LIN {X 0,Y 481.676,Z 380.486,A -85,B 0,C 180,E1 -6886.848,E2 -6886.848} C_VEL
LIN {X 0,Y 481.68,Z 380.488,A -85,B 0,C 180,E1 -6890.064,E2 -6890.064} C_VEL
LIN {X 0,Y 481.619,Z 380.495,A -85,B 0,C 180,E1 -6893.256,E2 -6893.256} C_VEL
LIN {X 0,Y 481.719,Z 380.64,A -85,B 0,C 180,E1 -6895.758,E2 -6895.758} C_VEL
LIN {X 0,Y 483.205,Z 388.494,A -85,B 0,C 180,E1 -6898.429,E2 -6898.429} C_VEL
LIN {X 0,Y 483.717,Z 393.145,A -85,B 0,C 180,E1 -6899.92,E2 -6899.92} C_VEL
LIN {X 0,Y 483.106,Z 403.096,A -85,B 0,C 180,E1 -6902.865,E2 -6902.865} C_VEL
LIN {X 0,Y 482.561,Z 413.944,A -85,B 0,C 180,E1 -6905.937,E2 -6905.937} C_VEL
LIN {X 0,Y 482.061,Z 425.792,A -85,B 0,C 180,E1 -6909.208,E2 -6909.208} C_VEL
LIN {X 0,Y 481.663,Z 438.463,A -85,B 0,C 180,E1 -6912.598,E2 -6912.598} C_VEL
LIN {X 0,Y 481.415,Z 448.444,A -85,B 0,C 180,E1 -6915.2,E2 -6915.2} C_VEL
LIN {X 0,Y 483.253,Z 462.341,A -85,B 0,C 180,E1 -6915.581,E2 -6915.581} C_VEL
LIN {X 0,Y 483.6,Z 467.954,A -85,B 0,C 180,E1 -6915.779,E2 -6915.779} C_VEL
LIN {X 0,Y 483.17,Z 480.671,A -85,B 0,C 180,E1 -6916.33,E2 -6916.33} C_VEL
LIN {X 0,Y 482.784,Z 492.217,A -85,B 0,C 180,E1 -6917.005,E2 -6917.005} C_VEL
LIN {X 0,Y 482.404,Z 503.568,A -85,B 0,C 180,E1 -6917.852,E2 -6917.852} C_VEL
LIN {X 0,Y 482.056,Z 513.298,A -85,B 0,C 180,E1 -6918.758,E2 -6918.758} C_VEL
LIN {X 0,Y 481.599,Z 523.341,A -85,B 0,C 180,E1 -6919.917,E2 -6919.917} C_VEL
LIN {X 0,Y 481.317,Z 532.179,A -85,B 0,C 180,E1 -6921.183,E2 -6921.183} C_VEL
LIN {X 0,Y 481.104,Z 539.214,A -85,B 0,C 180,E1 -6922.447,E2 -6922.447} C_VEL
LIN {X 0,Y 480.936,Z 545.233,A -85,B 0,C 180,E1 -6923.812,E2 -6923.812} C_VEL
LIN {X 0,Y 480.904,Z 549.252,A -85,B 0,C 180,E1 -6924.972,E2 -6924.972} C_VEL
LIN {X 0,Y 480.851,Z 551.584,A -85,B 0,C 180,E1 -6925.811,E2 -6925.811} C_VEL
LIN {X 0,Y 480.893,Z 553.484,A -85,B 0,C 180,E1 -6926.651,E2 -6926.651} C_VEL
LIN {X 0,Y 480.869,Z 554.904,A -85,B 0,C 180,E1 -6927.489,E2 -6927.489} C_VEL
LIN {X 0,Y 480.824,Z 555.914,A -85,B 0,C 180,E1 -6928.327,E2 -6928.327} C_VEL
LIN {X 0,Y 480.743,Z 556.751,A -85,B 0,C 180,E1 -6930.002,E2 -6930.002} C_VEL
LIN {X 0,Y 480.825,Z 555.927,A -85,B 0,C 180,E1 -6931.677,E2 -6931.677} C_VEL
LIN {X 0,Y 480.87,Z 554.926,A -85,B 0,C 180,E1 -6932.515,E2 -6932.515} C_VEL
LIN {X 0,Y 480.894,Z 553.512,A -85,B 0,C 180,E1 -6933.353,E2 -6933.353} C_VEL
LIN {X 0,Y 480.847,Z 550.542,A -85,B 0,C 180,E1 -6934.613,E2 -6934.613} C_VEL
LIN {X 0,Y 480.952,Z 546.523,A -85,B 0,C 180,E1 -6935.873,E2 -6935.873} C_VEL
LIN {X 0,Y 481.11,Z 540.312,A -85,B 0,C 180,E1 -6937.345,E2 -6937.345} C_VEL
LIN {X 0,Y 481.308,Z 533.534,A -85,B 0,C 180,E1 -6938.609,E2 -6938.609} C_VEL
LIN {X 0,Y 481.557,Z 525.1,A -85,B 0,C 180,E1 -6939.876,E2 -6939.876} C_VEL
LIN {X 0,Y 481.935,Z 516.392,A -85,B 0,C 180,E1 -6940.93,E2 -6940.93} C_VEL
LIN {X 0,Y 482.315,Z 505.902,A -85,B 0,C 180,E1 -6941.963,E2 -6941.963} C_VEL
LIN {X 0,Y 482.683,Z 495.234,A -85,B 0,C 180,E1 -6942.809,E2 -6942.809} C_VEL
LIN {X 0,Y 483.131,Z 482.915,A -85,B 0,C 180,E1 -6943.568,E2 -6943.568} C_VEL
LIN {X 0,Y 483.542,Z 470.344,A -85,B 0,C 180,E1 -6944.146,E2 -6944.146} C_VEL
LIN {X 0,Y 483.49,Z 464.03,A -85,B 0,C 180,E1 -6944.375,E2 -6944.375} C_VEL
LIN {X 0,Y 481.762,Z 451.22,A -85,B 0,C 180,E1 -6944.751,E2 -6944.751} C_VEL
LIN {X 0,Y 481.415,Z 448.546,A -85,B 0,C 180,E1 -6944.83,E2 -6944.83} C_VEL
LIN {X 0,Y 481.748,Z 435.725,A -85,B 0,C 180,E1 -6948.186,E2 -6948.186} C_VEL
LIN {X 0,Y 482.152,Z 423.863,A -85,B 0,C 180,E1 -6951.373,E2 -6951.373} C_VEL
LIN {X 0,Y 482.662,Z 412.396,A -85,B 0,C 180,E1 -6954.52,E2 -6954.52} C_VEL
LIN {X 0,Y 483.215,Z 401.049,A -85,B 0,C 180,E1 -6957.738,E2 -6957.738} C_VEL
LIN {X 0,Y 483.662,Z 393.005,A -85,B 0,C 180,E1 -6960.088,E2 -6960.088} C_VEL
LIN {X 0,Y 483.172,Z 388.19,A -85,B 0,C 180,E1 -6961.578,E2 -6961.578} C_VEL
LIN {X 0,Y 481.724,Z 380.48,A -85,B 0,C 180,E1 -6964.174,E2 -6964.174} C_VEL
LIN {X 0,Y 481.63,Z 380.493,A -85,B 0,C 180,E1 -6967.798,E2 -6967.798} C_VEL
LIN {X 0,Y 481.643,Z 380.488,A -85,B 0,C 180,E1 -6970.644,E2 -6970.644} C_VEL
LIN {X 0,Y 481.619,Z 380.494,A -85,B 0,C 180,E1 -6973.303,E2 -6973.303} C_VEL
LIN {X 0,Y 481.658,Z 380.486,A -85,B 0,C 180,E1 -6975.642,E2 -6975.642} C_VEL
LIN {X 0,Y 481.632,Z 380.49,A -85,B 0,C 180,E1 -6978.955,E2 -6978.955} C_VEL
LIN {X 0,Y 481.659,Z 380.484,A -85,B 0,C 180,E1 -6981.993,E2 -6981.993} C_VEL
LIN {X 0,Y 481.689,Z 380.481,A -85,B 0,C 180,E1 -6985.318,E2 -6985.318} C_VEL
LIN {X 0,Y 481.647,Z 380.488,A -85,B 0,C 180,E1 -6988.311,E2 -6988.311} C_VEL
LIN {X 0,Y 481.663,Z 380.488,A -85,B 0,C 180,E1 -6991.216,E2 -6991.216} C_VEL
LIN {X 0,Y 481.621,Z 380.49,A -85,B 0,C 180,E1 -6994.038,E2 -6994.038} C_VEL
LIN {X 0,Y 481.658,Z 380.491,A -85,B 0,C 180,E1 -6996.818,E2 -6996.818} C_VEL
LIN {X 0,Y 481.7,Z 380.481,A -85,B 0,C 180,E1 -6999.503,E2 -6999.503} C_VEL
LIN {X 0,Y 481.709,Z 380.485,A -85,B 0,C 180,E1 -7002.158,E2 -7002.158} C_VEL
LIN {X 0,Y 481.747,Z 380.476,A -85,B 0,C 180,E1 -7004.776,E2 -7004.776} C_VEL
LIN {X 0,Y 481.754,Z 380.476,A -85,B 0,C 180,E1 -7008.215,E2 -7008.215} C_VEL
LIN {X 0,Y 481.719,Z 380.481,A -85,B 0,C 180,E1 -7011.611,E2 -7011.611} C_VEL
LIN {X 0,Y 481.781,Z 380.473,A -85,B 0,C 180,E1 -7014.139,E2 -7014.139} C_VEL
LIN {X 0,Y 481.503,Z 380.649,A -85,B 0,C 180,E1 -7016.967,E2 -7016.967} C_VEL
LIN {X 0,Y 481.645,Z 387.989,A -85,B 0,C 180,E1 -7020,E2 -7020} C_VEL
LIN {X 0,Y 481.317,Z 393.994,A -85,B 0,C 180,E1 -7022.51,E2 -7022.51} C_VEL
LIN {X 0,Y 481.398,Z 399.763,A -85,B 0,C 180,E1 -7025.025,E2 -7025.025} C_VEL
LIN {X 0,Y 481.34,Z 405.639,A -85,B 0,C 180,E1 -7027.551,E2 -7027.551} C_VEL
LIN {X 0,Y 481.25,Z 413.309,A -85,B 0,C 180,E1 -7030.944,E2 -7030.944} C_VEL
LIN {X 0,Y 481.1,Z 420.994,A -85,B 0,C 180,E1 -7034.379,E2 -7034.379} C_VEL
LIN {X 0,Y 481.05,Z 424.92,A -85,B 0,C 180,E1 -7036.143,E2 -7036.143} C_VEL
LIN {X 0,Y 483.616,Z 438.35,A -85,B 0,C 180,E1 -7036.597,E2 -7036.597} C_VEL
LIN {X 0,Y 483.92,Z 441.544,A -85,B 0,C 180,E1 -7036.722,E2 -7036.722} C_VEL
LIN {X 0,Y 483.588,Z 454.148,A -85,B 0,C 180,E1 -7037.278,E2 -7037.278} C_VEL
LIN {X 0,Y 483.157,Z 464.801,A -85,B 0,C 180,E1 -7037.895,E2 -7037.895} C_VEL
LIN {X 0,Y 482.794,Z 475.459,A -85,B 0,C 180,E1 -7038.678,E2 -7038.678} C_VEL
LIN {X 0,Y 482.35,Z 486.451,A -85,B 0,C 180,E1 -7039.69,E2 -7039.69} C_VEL
LIN {X 0,Y 481.93,Z 495.839,A -85,B 0,C 180,E1 -7040.757,E2 -7040.757} C_VEL
LIN {X 0,Y 481.61,Z 503.654,A -85,B 0,C 180,E1 -7041.846,E2 -7041.846} C_VEL
LIN {X 0,Y 481.338,Z 511.583,A -85,B 0,C 180,E1 -7043.217,E2 -7043.217} C_VEL
LIN {X 0,Y 481.031,Z 517.926,A -85,B 0,C 180,E1 -7044.602,E2 -7044.602} C_VEL
LIN {X 0,Y 480.953,Z 522.785,A -85,B 0,C 180,E1 -7046,E2 -7046} C_VEL
LIN {X 0,Y 480.834,Z 526.37,A -85,B 0,C 180,E1 -7047.413,E2 -7047.413} C_VEL
LIN {X 0,Y 480.752,Z 528.76,A -85,B 0,C 180,E1 -7048.843,E2 -7048.843} C_VEL
LIN {X 0,Y 480.729,Z 530.029,A -85,B 0,C 180,E1 -7050.395,E2 -7050.395} C_VEL
LIN {X 0,Y 480.712,Z 529.851,A -85,B 0,C 180,E1 -7052.008,E2 -7052.008} C_VEL
LIN {X 0,Y 480.744,Z 528.314,A -85,B 0,C 180,E1 -7053.561,E2 -7053.561} C_VEL
LIN {X 0,Y 480.831,Z 525.481,A -85,B 0,C 180,E1 -7055.062,E2 -7055.062} C_VEL
LIN {X 0,Y 480.977,Z 521.357,A -85,B 0,C 180,E1 -7056.518,E2 -7056.518} C_VEL
LIN {X 0,Y 481.115,Z 516.002,A -85,B 0,C 180,E1 -7057.924,E2 -7057.924} C_VEL
LIN {X 0,Y 481.368,Z 509.214,A -85,B 0,C 180,E1 -7059.302,E2 -7059.302} C_VEL
LIN {X 0,Y 481.699,Z 500.773,A -85,B 0,C 180,E1 -7060.651,E2 -7060.651} C_VEL
LIN {X 0,Y 482.022,Z 492.106,A -85,B 0,C 180,E1 -7061.771,E2 -7061.771} C_VEL
LIN {X 0,Y 482.459,Z 482.471,A -85,B 0,C 180,E1 -7062.78,E2 -7062.78} C_VEL
LIN {X 0,Y 482.875,Z 471.084,A -85,B 0,C 180,E1 -7063.744,E2 -7063.744} C_VEL
LIN {X 0,Y 483.301,Z 460.089,A -85,B 0,C 180,E1 -7064.479,E2 -7064.479} C_VEL
LIN {X 0,Y 483.712,Z 448.856,A -85,B 0,C 180,E1 -7065.06,E2 -7065.06} C_VEL
LIN {X 0,Y 483.741,Z 439.076,A -85,B 0,C 180,E1 -7065.458,E2 -7065.458} C_VEL
LIN {X 0,Y 481.378,Z 426.409,A -85,B 0,C 180,E1 -7065.891,E2 -7065.891} C_VEL
LIN {X 0,Y 481.036,Z 424.605,A -85,B 0,C 180,E1 -7065.96,E2 -7065.96} C_VEL
LIN {X 0,Y 481.132,Z 418.161,A -85,B 0,C 180,E1 -7068.903,E2 -7068.903} C_VEL
LIN {X 0,Y 481.192,Z 411.015,A -85,B 0,C 180,E1 -7072.161,E2 -7072.161} C_VEL
LIN {X 0,Y 481.33,Z 404.161,A -85,B 0,C 180,E1 -7075.287,E2 -7075.287} C_VEL
LIN {X 0,Y 481.362,Z 403.419,A -85,B 0,C 180,E1 -7075.624,E2 -7075.624} C_VEL
LIN {X 0,Y 480.754,Z 402.002,A -85,B 0,C 180,E1 -7076.302,E2 -7076.302} C_VEL
LIN {X 0,Y 477.91,Z 399.902,A -85,B 0,C 180,E1 -7077.409,E2 -7077.409} C_VEL
LIN {X 0,Y 475.496,Z 398.224,A -85,B 0,C 180,E1 -7078.302,E2 -7078.302} C_VEL
LIN {X 0,Y 474.494,Z 396.844,A -85,B 0,C 180,E1 -7078.99,E2 -7078.99} C_VEL
LIN {X 0,Y 474.432,Z 396.349,A -85,B 0,C 180,E1 -7079.221,E2 -7079.221} C_VEL
LIN {X 0,Y 474.464,Z 389.854,A -85,B 0,C 180,E1 -7082.185,E2 -7082.185} C_VEL
LIN {X 0,Y 474.646,Z 382.584,A -85,B 0,C 180,E1 -7085.505,E2 -7085.505} C_VEL
LIN {X 0,Y 474.683,Z 381.36,A -85,B 0,C 180,E1 -7086.088,E2 -7086.088} C_VEL
LIN {X 0,Y 474.673,Z 381.359,A -85,B 0,C 180,E1 -7089.184,E2 -7089.184} C_VEL
LIN {X 0,Y 474.646,Z 381.364,A -85,B 0,C 180,E1 -7091.882,E2 -7091.882} C_VEL
LIN {X 0,Y 474.702,Z 381.353,A -85,B 0,C 180,E1 -7094.543,E2 -7094.543} C_VEL
LIN {X 0,Y 474.705,Z 381.355,A -85,B 0,C 180,E1 -7098.036,E2 -7098.036} C_VEL
LIN {X 0,Y 474.727,Z 381.355,A -85,B 0,C 180,E1 -7101.485,E2 -7101.485} C_VEL
LIN {X 0,Y 474.743,Z 381.352,A -85,B 0,C 180,E1 -7104.902,E2 -7104.902} C_VEL
LIN {X 0,Y 474.874,Z 381.335,A -85,B 0,C 180,E1 -7107.453,E2 -7107.453} C_VEL
LIN {X 0,Y 474.91,Z 381.45,A -85,B 0,C 180,E1 -7109.892,E2 -7109.892} C_VEL
LIN {X 0,Y 474.733,Z 386.231,A -85,B 0,C 180,E1 -7112.544,E2 -7112.544} C_VEL
LIN {X 0,Y 474.574,Z 392.513,A -85,B 0,C 180,E1 -7115.948,E2 -7115.948} C_VEL
LIN {X 0,Y 474.425,Z 397.306,A -85,B 0,C 180,E1 -7118.517,E2 -7118.517} C_VEL
LIN {X 0,Y 474.306,Z 403.992,A -85,B 0,C 180,E1 -7122.056,E2 -7122.056} C_VEL
LIN {X 0,Y 474.1,Z 410.649,A -85,B 0,C 180,E1 -7125.518,E2 -7125.518} C_VEL
LIN {X 0,Y 473.939,Z 417.514,A -85,B 0,C 180,E1 -7129.038,E2 -7129.038} C_VEL
LIN {X 0,Y 473.922,Z 421.247,A -85,B 0,C 180,E1 -7130.937,E2 -7130.937} C_VEL
LIN {X 0,Y 475.816,Z 432.165,A -85,B 0,C 180,E1 -7131.36,E2 -7131.36} C_VEL
LIN {X 0,Y 476.036,Z 438.597,A -85,B 0,C 180,E1 -7131.657,E2 -7131.657} C_VEL
LIN {X 0,Y 475.665,Z 448.951,A -85,B 0,C 180,E1 -7132.245,E2 -7132.245} C_VEL
LIN {X 0,Y 475.314,Z 458.419,A -85,B 0,C 180,E1 -7132.951,E2 -7132.951} C_VEL
LIN {X 0,Y 474.982,Z 468.268,A -85,B 0,C 180,E1 -7133.892,E2 -7133.892} C_VEL
LIN {X 0,Y 474.64,Z 477.014,A -85,B 0,C 180,E1 -7134.958,E2 -7134.958} C_VEL
LIN {X 0,Y 474.346,Z 484.62,A -85,B 0,C 180,E1 -7136.151,E2 -7136.151} C_VEL
LIN {X 0,Y 474.047,Z 490.599,A -85,B 0,C 180,E1 -7137.358,E2 -7137.358} C_VEL
LIN {X 0,Y 473.984,Z 495.44,A -85,B 0,C 180,E1 -7138.65,E2 -7138.65} C_VEL
LIN {X 0,Y 473.866,Z 498.551,A -85,B 0,C 180,E1 -7139.788,E2 -7139.788} C_VEL
LIN {X 0,Y 473.714,Z 501.15,A -85,B 0,C 180,E1 -7141.279,E2 -7141.279} C_VEL
LIN {X 0,Y 473.679,Z 502.019,A -85,B 0,C 180,E1 -7142.282,E2 -7142.282} C_VEL
LIN {X 0,Y 473.693,Z 502.038,A -85,B 0,C 180,E1 -7143.814,E2 -7143.814} C_VEL
LIN {X 0,Y 473.799,Z 500.472,A -85,B 0,C 180,E1 -7145.342,E2 -7145.342} C_VEL
LIN {X 0,Y 473.948,Z 497.426,A -85,B 0,C 180,E1 -7146.799,E2 -7146.799} C_VEL
LIN {X 0,Y 474.043,Z 494.299,A -85,B 0,C 180,E1 -7147.824,E2 -7147.824} C_VEL
LIN {X 0,Y 474.216,Z 489.417,A -85,B 0,C 180,E1 -7149.036,E2 -7149.036} C_VEL
LIN {X 0,Y 474.438,Z 483.837,A -85,B 0,C 180,E1 -7150.115,E2 -7150.115} C_VEL
LIN {X 0,Y 474.683,Z 477.63,A -85,B 0,C 180,E1 -7151.084,E2 -7151.084} C_VEL
LIN {X 0,Y 474.927,Z 470.21,A -85,B 0,C 180,E1 -7152.025,E2 -7152.025} C_VEL
LIN {X 0,Y 475.324,Z 460.576,A -85,B 0,C 180,E1 -7152.993,E2 -7152.993} C_VEL
LIN {X 0,Y 475.726,Z 451.213,A -85,B 0,C 180,E1 -7153.726,E2 -7153.726} C_VEL
LIN {X 0,Y 476.046,Z 440.21,A -85,B 0,C 180,E1 -7154.39,E2 -7154.39} C_VEL
LIN {X 0,Y 475.974,Z 432.535,A -85,B 0,C 180,E1 -7154.746,E2 -7154.746} C_VEL
LIN {X 0,Y 473.94,Z 421.51,A -85,B 0,C 180,E1 -7155.188,E2 -7155.188} C_VEL
LIN {X 0,Y 474.031,Z 415.761,A -85,B 0,C 180,E1 -7158.151,E2 -7158.151} C_VEL
LIN {X 0,Y 474.098,Z 409.341,A -85,B 0,C 180,E1 -7161.494,E2 -7161.494} C_VEL
LIN {X 0,Y 474.207,Z 405.279,A -85,B 0,C 180,E1 -7163.643,E2 -7163.643} C_VEL
LIN {X 0,Y 474.346,Z 399.44,A -85,B 0,C 180,E1 -7166.757,E2 -7166.757} C_VEL
LIN {X 0,Y 474.483,Z 393.793,A -85,B 0,C 180,E1 -7169.762,E2 -7169.762} C_VEL
LIN {X 0,Y 474.692,Z 388.447,A -85,B 0,C 180,E1 -7172.68,E2 -7172.68} C_VEL
LIN {X 0,Y 474.819,Z 383.281,A -85,B 0,C 180,E1 -7175.516,E2 -7175.516} C_VEL
LIN {X 0,Y 474.697,Z 381.36,A -85,B 0,C 180,E1 -7176.617,E2 -7176.617} C_VEL
LIN {X 0,Y 474.633,Z 381.365,A -85,B 0,C 180,E1 -7180.089,E2 -7180.089} C_VEL
LIN {X 0,Y 474.627,Z 381.367,A -85,B 0,C 180,E1 -7182.774,E2 -7182.774} C_VEL
LIN {X 0,Y 474.63,Z 381.365,A -85,B 0,C 180,E1 -7185.421,E2 -7185.421} C_VEL
LIN {X 0,Y 474.719,Z 381.353,A -85,B 0,C 180,E1 -7188.038,E2 -7188.038} C_VEL
LIN {X 0,Y 474.711,Z 381.355,A -85,B 0,C 180,E1 -7191.486,E2 -7191.486} C_VEL
LIN {X 0,Y 474.769,Z 381.348,A -85,B 0,C 180,E1 -7194.053,E2 -7194.053} C_VEL
LIN {X 0,Y 474.88,Z 381.333,A -85,B 0,C 180,E1 -7197.456,E2 -7197.456} C_VEL
LIN {X 0,Y 474.886,Z 381.332,A -85,B 0,C 180,E1 -7200,E2 -7200} C_VEL
LIN {X 0,Y 474.88,Z 381.332,A -85,B 0,C 180,E1 -7202.545,E2 -7202.545} C_VEL
LIN {X 0,Y 474.77,Z 381.347,A -85,B 0,C 180,E1 -7205.948,E2 -7205.948} C_VEL
LIN {X 0,Y 474.707,Z 381.357,A -85,B 0,C 180,E1 -7208.514,E2 -7208.514} C_VEL
LIN {X 0,Y 474.72,Z 381.351,A -85,B 0,C 180,E1 -7211.962,E2 -7211.962} C_VEL
LIN {X 0,Y 474.68,Z 381.356,A -85,B 0,C 180,E1 -7215.779,E2 -7215.779} C_VEL
LIN {X 0,Y 474.646,Z 381.36,A -85,B 0,C 180,E1 -7219.011,E2 -7219.011} C_VEL
LIN {X 0,Y 474.623,Z 381.363,A -85,B 0,C 180,E1 -7221.728,E2 -7221.728} C_VEL
LIN {X 0,Y 474.641,Z 381.361,A -85,B 0,C 180,E1 -7224.494,E2 -7224.494} C_VEL
LIN {X 0,Y 474.678,Z 381.357,A -85,B 0,C 180,E1 -7227.34,E2 -7227.34} C_VEL
LIN {X 0,Y 474.59,Z 381.368,A -85,B 0,C 180,E1 -7230.813,E2 -7230.813} C_VEL
LIN {X 0,Y 474.62,Z 381.367,A -85,B 0,C 180,E1 -7233.986,E2 -7233.986} C_VEL
LIN {X 0,Y 474.559,Z 381.375,A -85,B 0,C 180,E1 -7236.902,E2 -7236.902} C_VEL
LIN {X 0,Y 474.638,Z 381.364,A -85,B 0,C 180,E1 -7239.654,E2 -7239.654} C_VEL
LIN {X 0,Y 474.637,Z 381.364,A -85,B 0,C 180,E1 -7242.932,E2 -7242.932} C_VEL
LIN {X 0,Y 474.604,Z 381.368,A -85,B 0,C 180,E1 -7245.898,E2 -7245.898} C_VEL
LIN {X 0,Y 474.633,Z 381.365,A -85,B 0,C 180,E1 -7249.041,E2 -7249.041} C_VEL
LIN {X 0,Y 474.608,Z 381.368,A -85,B 0,C 180,E1 -7251.705,E2 -7251.705} C_VEL
LIN {X 0,Y 474.653,Z 381.381,A -85,B 0,C 180,E1 -7255.394,E2 -7255.394} C_VEL
LIN {X 0,Y 476.288,Z 390.069,A -85,B 0,C 180,E1 -7258.409,E2 -7258.409} C_VEL
LIN {X 0,Y 476.747,Z 394.694,A -85,B 0,C 180,E1 -7259.923,E2 -7259.923} C_VEL
LIN {X 0,Y 476.124,Z 404.14,A -85,B 0,C 180,E1 -7262.771,E2 -7262.771} C_VEL
LIN {X 0,Y 475.535,Z 415.372,A -85,B 0,C 180,E1 -7266.023,E2 -7266.023} C_VEL
LIN {X 0,Y 475.017,Z 426.749,A -85,B 0,C 180,E1 -7269.204,E2 -7269.204} C_VEL
LIN {X 0,Y 474.614,Z 438.219,A -85,B 0,C 180,E1 -7272.331,E2 -7272.331} C_VEL
LIN {X 0,Y 474.366,Z 448.416,A -85,B 0,C 180,E1 -7275.003,E2 -7275.003} C_VEL
LIN {X 0,Y 476.165,Z 462.258,A -85,B 0,C 180,E1 -7275.389,E2 -7275.389} C_VEL
LIN {X 0,Y 476.669,Z 467.857,A -85,B 0,C 180,E1 -7275.596,E2 -7275.596} C_VEL
LIN {X 0,Y 476.268,Z 480.007,A -85,B 0,C 180,E1 -7276.128,E2 -7276.128} C_VEL
LIN {X 0,Y 475.802,Z 492.581,A -85,B 0,C 180,E1 -7276.876,E2 -7276.876} C_VEL
LIN {X 0,Y 475.375,Z 503.595,A -85,B 0,C 180,E1 -7277.718,E2 -7277.718} C_VEL
LIN {X 0,Y 475.005,Z 513.788,A -85,B 0,C 180,E1 -7278.697,E2 -7278.697} C_VEL
LIN {X 0,Y 474.562,Z 522.866,A -85,B 0,C 180,E1 -7279.766,E2 -7279.766} C_VEL
LIN {X 0,Y 474.258,Z 531.723,A -85,B 0,C 180,E1 -7281.051,E2 -7281.051} C_VEL
LIN {X 0,Y 474.034,Z 538.776,A -85,B 0,C 180,E1 -7282.334,E2 -7282.334} C_VEL
LIN {X 0,Y 473.848,Z 544.281,A -85,B 0,C 180,E1 -7283.582,E2 -7283.582} C_VEL
LIN {X 0,Y 473.838,Z 548.833,A -85,B 0,C 180,E1 -7284.896,E2 -7284.896} C_VEL
LIN {X 0,Y 473.754,Z 551.167,A -85,B 0,C 180,E1 -7285.748,E2 -7285.748} C_VEL
LIN {X 0,Y 473.819,Z 553.072,A -85,B 0,C 180,E1 -7286.601,E2 -7286.601} C_VEL
LIN {X 0,Y 473.783,Z 554.495,A -85,B 0,C 180,E1 -7287.451,E2 -7287.451} C_VEL
LIN {X 0,Y 473.758,Z 555.508,A -85,B 0,C 180,E1 -7288.302,E2 -7288.302} C_VEL
LIN {X 0,Y 473.67,Z 556.348,A -85,B 0,C 180,E1 -7290.002,E2 -7290.002} C_VEL
LIN {X 0,Y 473.758,Z 555.525,A -85,B 0,C 180,E1 -7291.702,E2 -7291.702} C_VEL
LIN {X 0,Y 473.784,Z 554.522,A -85,B 0,C 180,E1 -7292.552,E2 -7292.552} C_VEL
LIN {X 0,Y 473.82,Z 553.106,A -85,B 0,C 180,E1 -7293.403,E2 -7293.403} C_VEL
LIN {X 0,Y 473.77,Z 550.134,A -85,B 0,C 180,E1 -7294.682,E2 -7294.682} C_VEL
LIN {X 0,Y 473.856,Z 546.108,A -85,B 0,C 180,E1 -7295.961,E2 -7295.961} C_VEL
LIN {X 0,Y 474.019,Z 539.889,A -85,B 0,C 180,E1 -7297.456,E2 -7297.456} C_VEL
LIN {X 0,Y 474.235,Z 533.101,A -85,B 0,C 180,E1 -7298.739,E2 -7298.739} C_VEL
LIN {X 0,Y 474.497,Z 524.644,A -85,B 0,C 180,E1 -7300.024,E2 -7300.024} C_VEL
LIN {X 0,Y 474.892,Z 515.912,A -85,B 0,C 180,E1 -7301.094,E2 -7301.094} C_VEL
LIN {X 0,Y 475.283,Z 505.622,A -85,B 0,C 180,E1 -7302.121,E2 -7302.121} C_VEL
LIN {X 0,Y 475.737,Z 494.376,A -85,B 0,C 180,E1 -7303.021,E2 -7303.021} C_VEL
LIN {X 0,Y 476.195,Z 482.263,A -85,B 0,C 180,E1 -7303.769,E2 -7303.769} C_VEL
LIN {X 0,Y 476.613,Z 469.574,A -85,B 0,C 180,E1 -7304.356,E2 -7304.356} C_VEL
LIN {X 0,Y 476.524,Z 464.706,A -85,B 0,C 180,E1 -7304.536,E2 -7304.536} C_VEL
LIN {X 0,Y 474.842,Z 451.844,A -85,B 0,C 180,E1 -7304.934,E2 -7304.934} C_VEL
LIN {X 0,Y 474.366,Z 448.348,A -85,B 0,C 180,E1 -7305.028,E2 -7305.028} C_VEL
LIN {X 0,Y 474.71,Z 435.803,A -85,B 0,C 180,E1 -7308.387,E2 -7308.387} C_VEL
LIN {X 0,Y 475.154,Z 423.664,A -85,B 0,C 180,E1 -7311.703,E2 -7311.703} C_VEL
LIN {X 0,Y 475.712,Z 412.251,A -85,B 0,C 180,E1 -7314.902,E2 -7314.902} C_VEL
LIN {X 0,Y 476.342,Z 400.942,A -85,B 0,C 180,E1 -7318.174,E2 -7318.174} C_VEL
LIN {X 0,Y 476.705,Z 394.535,A -85,B 0,C 180,E1 -7320.085,E2 -7320.085} C_VEL
LIN {X 0,Y 476.251,Z 389.742,A -85,B 0,C 180,E1 -7321.593,E2 -7321.593} C_VEL
LIN {X 0,Y 474.685,Z 381.356,A -85,B 0,C 180,E1 -7324.431,E2 -7324.431} C_VEL
LIN {X 0,Y 474.591,Z 381.368,A -85,B 0,C 180,E1 -7327.385,E2 -7327.385} C_VEL
LIN {X 0,Y 474.611,Z 381.368,A -85,B 0,C 180,E1 -7329.645,E2 -7329.645} C_VEL
LIN {X 0,Y 474.571,Z 381.37,A -85,B 0,C 180,E1 -7332.94,E2 -7332.94} C_VEL
LIN {X 0,Y 474.608,Z 381.361,A -85,B 0,C 180,E1 -7335.895,E2 -7335.895} C_VEL
LIN {X 0,Y 474.607,Z 381.365,A -85,B 0,C 180,E1 -7339.045,E2 -7339.045} C_VEL
LIN {X 0,Y 474.615,Z 381.36,A -85,B 0,C 180,E1 -7341.705,E2 -7341.705} C_VEL
LIN {X 0,Y 474.629,Z 381.363,A -85,B 0,C 180,E1 -7344.726,E2 -7344.726} C_VEL
LIN {X 0,Y 474.633,Z 381.365,A -85,B 0,C 180,E1 -7347.787,E2 -7347.787} C_VEL
LIN {X 0,Y 474.603,Z 381.365,A -85,B 0,C 180,E1 -7350.891,E2 -7350.891} C_VEL
LIN {X 0,Y 474.575,Z 381.371,A -85,B 0,C 180,E1 -7353.623,E2 -7353.623} C_VEL
LIN {X 0,Y 474.639,Z 381.363,A -85,B 0,C 180,E1 -7356.642,E2 -7356.642} C_VEL
LIN {X 0,Y 474.659,Z 381.36,A -85,B 0,C 180,E1 -7360.089,E2 -7360.089} C_VEL
LIN {X 0,Y 474.653,Z 381.361,A -85,B 0,C 180,E1 -7362.774,E2 -7362.774} C_VEL
LIN {X 0,Y 474.651,Z 381.362,A -85,B 0,C 180,E1 -7365.421,E2 -7365.421} C_VEL
LIN {X 0,Y 474.708,Z 381.355,A -85,B 0,C 180,E1 -7368.037,E2 -7368.037} C_VEL
LIN {X 0,Y 474.669,Z 381.361,A -85,B 0,C 180,E1 -7371.485,E2 -7371.485} C_VEL
LIN {X 0,Y 474.744,Z 381.349,A -85,B 0,C 180,E1 -7374.052,E2 -7374.052} C_VEL
LIN {X 0,Y 474.572,Z 381.371,A -85,B 0,C 180,E1 -7375.753,E2 -7375.753} C_VEL
LIN {X 0,Y 474.482,Z 381.56,A -85,B 0,C 180,E1 -7376.922,E2 -7376.922} C_VEL
LIN {X 0,Y 474.627,Z 387.942,A -85,B 0,C 180,E1 -7379.576,E2 -7379.576} C_VEL
LIN {X 0,Y 474.345,Z 393.996,A -85,B 0,C 180,E1 -7382.122,E2 -7382.122} C_VEL
LIN {X 0,Y 474.348,Z 400.847,A -85,B 0,C 180,E1 -7385.1,E2 -7385.1} C_VEL
LIN {X 0,Y 474.278,Z 406.608,A -85,B 0,C 180,E1 -7387.664,E2 -7387.664} C_VEL
LIN {X 0,Y 474.198,Z 414.433,A -85,B 0,C 180,E1 -7391.108,E2 -7391.108} C_VEL
LIN {X 0,Y 474.029,Z 422.187,A -85,B 0,C 180,E1 -7394.598,E2 -7394.598} C_VEL
LIN {X 0,Y 473.98,Z 425.118,A -85,B 0,C 180,E1 -7395.921,E2 -7395.921} C_VEL
LIN {X 0,Y 476.607,Z 438.496,A -85,B 0,C 180,E1 -7396.38,E2 -7396.38} C_VEL
LIN {X 0,Y 477.035,Z 442.309,A -85,B 0,C 180,E1 -7396.536,E2 -7396.536} C_VEL
LIN {X 0,Y 476.662,Z 454.69,A -85,B 0,C 180,E1 -7397.095,E2 -7397.095} C_VEL
LIN {X 0,Y 476.176,Z 466.887,A -85,B 0,C 180,E1 -7397.833,E2 -7397.833} C_VEL
LIN {X 0,Y 475.702,Z 478.517,A -85,B 0,C 180,E1 -7398.743,E2 -7398.743} C_VEL
LIN {X 0,Y 475.259,Z 488.977,A -85,B 0,C 180,E1 -7399.771,E2 -7399.771} C_VEL
LIN {X 0,Y 474.879,Z 497.525,A -85,B 0,C 180,E1 -7400.805,E2 -7400.805} C_VEL
LIN {X 0,Y 474.516,Z 505.394,A -85,B 0,C 180,E1 -7401.961,E2 -7401.961} C_VEL
LIN {X 0,Y 474.258,Z 512.538,A -85,B 0,C 180,E1 -7403.251,E2 -7403.251} C_VEL
LIN {X 0,Y 473.959,Z 518.215,A -85,B 0,C 180,E1 -7404.531,E2 -7404.531} C_VEL
LIN {X 0,Y 473.864,Z 523.034,A -85,B 0,C 180,E1 -7405.946,E2 -7405.946} C_VEL
LIN {X 0,Y 473.761,Z 526.6,A -85,B 0,C 180,E1 -7407.378,E2 -7407.378} C_VEL
LIN {X 0,Y 473.65,Z 529.07,A -85,B 0,C 180,E1 -7408.902,E2 -7408.902} C_VEL
LIN {X 0,Y 473.623,Z 530.264,A -85,B 0,C 180,E1 -7410.609,E2 -7410.609} C_VEL
LIN {X 0,Y 473.618,Z 529.888,A -85,B 0,C 180,E1 -7412.29,E2 -7412.29} C_VEL
LIN {X 0,Y 473.671,Z 528.193,A -85,B 0,C 180,E1 -7413.809,E2 -7413.809} C_VEL
LIN {X 0,Y 473.776,Z 525.105,A -85,B 0,C 180,E1 -7415.347,E2 -7415.347} C_VEL
LIN {X 0,Y 473.934,Z 520.883,A -85,B 0,C 180,E1 -7416.795,E2 -7416.795} C_VEL
LIN {X 0,Y 474.115,Z 515.332,A -85,B 0,C 180,E1 -7418.219,E2 -7418.219} C_VEL
LIN {X 0,Y 474.359,Z 508.331,A -85,B 0,C 180,E1 -7419.607,E2 -7419.607} C_VEL
LIN {X 0,Y 474.695,Z 500.77,A -85,B 0,C 180,E1 -7420.813,E2 -7420.813} C_VEL
LIN {X 0,Y 475.097,Z 491.316,A -85,B 0,C 180,E1 -7422.032,E2 -7422.032} C_VEL
LIN {X 0,Y 475.571,Z 480.833,A -85,B 0,C 180,E1 -7423.116,E2 -7423.116} C_VEL
LIN {X 0,Y 475.962,Z 470.939,A -85,B 0,C 180,E1 -7423.947,E2 -7423.947} C_VEL
LIN {X 0,Y 476.394,Z 459.562,A -85,B 0,C 180,E1 -7424.709,E2 -7424.709} C_VEL
LIN {X 0,Y 476.881,Z 447.37,A -85,B 0,C 180,E1 -7425.331,E2 -7425.331} C_VEL
LIN {X 0,Y 476.91,Z 440.464,A -85,B 0,C 180,E1 -7425.616,E2 -7425.616} C_VEL
LIN {X 0,Y 474.565,Z 427.858,A -85,B 0,C 180,E1 -7426.073,E2 -7426.073} C_VEL
LIN {X 0,Y 473.959,Z 424.803,A -85,B 0,C 180,E1 -7426.16,E2 -7426.16} C_VEL
LIN {X 0,Y 474.084,Z 417.992,A -85,B 0,C 180,E1 -7429.286,E2 -7429.286} C_VEL
LIN {X 0,Y 474.155,Z 410.839,A -85,B 0,C 180,E1 -7432.575,E2 -7432.575} C_VEL
LIN {X 0,Y 474.333,Z 403.954,A -85,B 0,C 180,E1 -7435.733,E2 -7435.733} C_VEL
LIN {X 0,Y 474.432,Z 396.349,A -85,B 0,C 180,E1 -7439.221,E2 -7439.221} C_VEL
LIN {X 0,Y 473.815,Z 394.927,A -85,B 0,C 180,E1 -7439.909,E2 -7439.909} C_VEL
LIN {X 0,Y 470.963,Z 392.816,A -85,B 0,C 180,E1 -7441.032,E2 -7441.032} C_VEL
LIN {X 0,Y 468.528,Z 391.146,A -85,B 0,C 180,E1 -7441.938,E2 -7441.938} C_VEL
LIN {X 0,Y 467.491,Z 389.773,A -85,B 0,C 180,E1 -7442.635,E2 -7442.635} C_VEL
LIN {X 0,Y 467.414,Z 389.278,A -85,B 0,C 180,E1 -7442.87,E2 -7442.87} C_VEL
LIN {X 0,Y 467.662,Z 382.234,A -85,B 0,C 180,E1 -7446.186,E2 -7446.186} C_VEL
LIN {X 0,Y 467.624,Z 382.235,A -85,B 0,C 180,E1 -7449.776,E2 -7449.776} C_VEL
LIN {X 0,Y 467.597,Z 382.239,A -85,B 0,C 180,E1 -7452.505,E2 -7452.505} C_VEL
LIN {X 0,Y 467.608,Z 382.241,A -85,B 0,C 180,E1 -7455.195,E2 -7455.195} C_VEL
LIN {X 0,Y 467.657,Z 382.232,A -85,B 0,C 180,E1 -7457.853,E2 -7457.853} C_VEL
LIN {X 0,Y 467.68,Z 382.232,A -85,B 0,C 180,E1 -7461.356,E2 -7461.356} C_VEL
LIN {X 0,Y 467.72,Z 382.225,A -85,B 0,C 180,E1 -7463.961,E2 -7463.961} C_VEL
LIN {X 0,Y 467.814,Z 382.214,A -85,B 0,C 180,E1 -7467.415,E2 -7467.415} C_VEL
LIN {X 0,Y 467.881,Z 382.272,A -85,B 0,C 180,E1 -7469.783,E2 -7469.783} C_VEL
LIN {X 0,Y 467.734,Z 385.754,A -85,B 0,C 180,E1 -7471.72,E2 -7471.72} C_VEL
LIN {X 0,Y 467.617,Z 391.977,A -85,B 0,C 180,E1 -7475.172,E2 -7475.172} C_VEL
LIN {X 0,Y 467.363,Z 398.391,A -85,B 0,C 180,E1 -7478.647,E2 -7478.647} C_VEL
LIN {X 0,Y 467.245,Z 404.964,A -85,B 0,C 180,E1 -7482.154,E2 -7482.154} C_VEL
LIN {X 0,Y 467.02,Z 411.736,A -85,B 0,C 180,E1 -7485.714,E2 -7485.714} C_VEL
LIN {X 0,Y 466.845,Z 418.732,A -85,B 0,C 180,E1 -7489.339,E2 -7489.339} C_VEL
LIN {X 0,Y 466.845,Z 421.429,A -85,B 0,C 180,E1 -7490.729,E2 -7490.729} C_VEL
LIN {X 0,Y 468.927,Z 433.19,A -85,B 0,C 180,E1 -7491.204,E2 -7491.204} C_VEL
LIN {X 0,Y 469.092,Z 439.11,A -85,B 0,C 180,E1 -7491.483,E2 -7491.483} C_VEL
LIN {X 0,Y 468.703,Z 450.105,A -85,B 0,C 180,E1 -7492.129,E2 -7492.129} C_VEL
LIN {X 0,Y 468.346,Z 459.412,A -85,B 0,C 180,E1 -7492.845,E2 -7492.845} C_VEL
LIN {X 0,Y 467.991,Z 468.583,A -85,B 0,C 180,E1 -7493.742,E2 -7493.742} C_VEL
LIN {X 0,Y 467.707,Z 475.981,A -85,B 0,C 180,E1 -7494.642,E2 -7494.642} C_VEL
LIN {X 0,Y 467.41,Z 482.17,A -85,B 0,C 180,E1 -7495.557,E2 -7495.557} C_VEL
LIN {X 0,Y 467.232,Z 487.819,A -85,B 0,C 180,E1 -7496.58,E2 -7496.58} C_VEL
LIN {X 0,Y 467.031,Z 493.124,A -85,B 0,C 180,E1 -7497.804,E2 -7497.804} C_VEL
LIN {X 0,Y 466.9,Z 497.586,A -85,B 0,C 180,E1 -7499.186,E2 -7499.186} C_VEL
LIN {X 0,Y 466.802,Z 499.051,A -85,B 0,C 180,E1 -7499.788,E2 -7499.788} C_VEL
LIN {X 0,Y 466.684,Z 501.037,A -85,B 0,C 180,E1 -7500.865,E2 -7500.865} C_VEL
LIN {X 0,Y 466.597,Z 502.121,A -85,B 0,C 180,E1 -7501.812,E2 -7501.812} C_VEL
LIN {X 0,Y 466.587,Z 502.615,A -85,B 0,C 180,E1 -7502.834,E2 -7502.834} C_VEL
LIN {X 0,Y 466.634,Z 502.313,A -85,B 0,C 180,E1 -7504.07,E2 -7504.07} C_VEL
LIN {X 0,Y 466.751,Z 500.51,A -85,B 0,C 180,E1 -7505.601,E2 -7505.601} C_VEL
LIN {X 0,Y 466.908,Z 497.222,A -85,B 0,C 180,E1 -7507.083,E2 -7507.083} C_VEL
LIN {X 0,Y 467.083,Z 492.441,A -85,B 0,C 180,E1 -7508.518,E2 -7508.518} C_VEL
LIN {X 0,Y 467.32,Z 485.988,A -85,B 0,C 180,E1 -7509.916,E2 -7509.916} C_VEL
LIN {X 0,Y 467.613,Z 479.068,A -85,B 0,C 180,E1 -7511.062,E2 -7511.062} C_VEL
LIN {X 0,Y 467.904,Z 471.348,A -85,B 0,C 180,E1 -7512.084,E2 -7512.084} C_VEL
LIN {X 0,Y 468.362,Z 461.659,A -85,B 0,C 180,E1 -7513.089,E2 -7513.089} C_VEL
LIN {X 0,Y 468.778,Z 451.607,A -85,B 0,C 180,E1 -7513.9,E2 -7513.9} C_VEL
LIN {X 0,Y 469.14,Z 440.242,A -85,B 0,C 180,E1 -7514.593,E2 -7514.593} C_VEL
LIN {X 0,Y 469.001,Z 433.224,A -85,B 0,C 180,E1 -7514.928,E2 -7514.928} C_VEL
LIN {X 0,Y 466.858,Z 421.765,A -85,B 0,C 180,E1 -7515.403,E2 -7515.403} C_VEL
LIN {X 0,Y 466.941,Z 417.689,A -85,B 0,C 180,E1 -7517.515,E2 -7517.515} C_VEL
LIN {X 0,Y 467.027,Z 411.438,A -85,B 0,C 180,E1 -7520.8,E2 -7520.8} C_VEL
LIN {X 0,Y 467.14,Z 407.274,A -85,B 0,C 180,E1 -7523.002,E2 -7523.002} C_VEL
LIN {X 0,Y 467.278,Z 401.396,A -85,B 0,C 180,E1 -7526.187,E2 -7526.187} C_VEL
LIN {X 0,Y 467.433,Z 395.699,A -85,B 0,C 180,E1 -7529.257,E2 -7529.257} C_VEL
LIN {X 0,Y 467.619,Z 389.87,A -85,B 0,C 180,E1 -7532.458,E2 -7532.458} C_VEL
LIN {X 0,Y 467.781,Z 385.072,A -85,B 0,C 180,E1 -7535.123,E2 -7535.123} C_VEL
LIN {X 0,Y 467.643,Z 382.239,A -85,B 0,C 180,E1 -7536.856,E2 -7536.856} C_VEL
LIN {X 0,Y 467.602,Z 382.241,A -85,B 0,C 180,E1 -7539.777,E2 -7539.777} C_VEL
LIN {X 0,Y 467.585,Z 382.244,A -85,B 0,C 180,E1 -7542.506,E2 -7542.506} C_VEL
LIN {X 0,Y 467.587,Z 382.243,A -85,B 0,C 180,E1 -7545.196,E2 -7545.196} C_VEL
LIN {X 0,Y 467.676,Z 382.23,A -85,B 0,C 180,E1 -7547.855,E2 -7547.855} C_VEL
LIN {X 0,Y 467.664,Z 382.234,A -85,B 0,C 180,E1 -7551.357,E2 -7551.357} C_VEL
LIN {X 0,Y 467.731,Z 382.225,A -85,B 0,C 180,E1 -7553.963,E2 -7553.963} C_VEL
LIN {X 0,Y 467.846,Z 382.209,A -85,B 0,C 180,E1 -7557.417,E2 -7557.417} C_VEL
LIN {X 0,Y 467.857,Z 382.207,A -85,B 0,C 180,E1 -7560,E2 -7560} C_VEL
LIN {X 0,Y 467.846,Z 382.209,A -85,B 0,C 180,E1 -7562.583,E2 -7562.583} C_VEL
LIN {X 0,Y 467.732,Z 382.223,A -85,B 0,C 180,E1 -7566.038,E2 -7566.038} C_VEL
LIN {X 0,Y 467.66,Z 382.233,A -85,B 0,C 180,E1 -7568.643,E2 -7568.643} C_VEL
LIN {X 0,Y 467.677,Z 382.229,A -85,B 0,C 180,E1 -7572.145,E2 -7572.145} C_VEL
LIN {X 0,Y 467.644,Z 382.232,A -85,B 0,C 180,E1 -7575.895,E2 -7575.895} C_VEL
LIN {X 0,Y 467.603,Z 382.239,A -85,B 0,C 180,E1 -7579.309,E2 -7579.309} C_VEL
LIN {X 0,Y 467.553,Z 382.246,A -85,B 0,C 180,E1 -7582.073,E2 -7582.073} C_VEL
LIN {X 0,Y 467.585,Z 382.243,A -85,B 0,C 180,E1 -7584.889,E2 -7584.889} C_VEL
LIN {X 0,Y 467.608,Z 382.238,A -85,B 0,C 180,E1 -7587.77,E2 -7587.77} C_VEL
LIN {X 0,Y 467.553,Z 382.245,A -85,B 0,C 180,E1 -7591.048,E2 -7591.048} C_VEL
LIN {X 0,Y 467.572,Z 382.244,A -85,B 0,C 180,E1 -7594.245,E2 -7594.245} C_VEL
LIN {X 0,Y 467.534,Z 382.248,A -85,B 0,C 180,E1 -7597.189,E2 -7597.189} C_VEL
LIN {X 0,Y 467.581,Z 382.242,A -85,B 0,C 180,E1 -7600.265,E2 -7600.265} C_VEL
LIN {X 0,Y 467.604,Z 382.239,A -85,B 0,C 180,E1 -7602.574,E2 -7602.574} C_VEL
LIN {X 0,Y 467.561,Z 382.247,A -85,B 0,C 180,E1 -7606.179,E2 -7606.179} C_VEL
LIN {X 0,Y 467.577,Z 382.244,A -85,B 0,C 180,E1 -7608.724,E2 -7608.724} C_VEL
LIN {X 0,Y 467.566,Z 382.246,A -85,B 0,C 180,E1 -7611.409,E2 -7611.409} C_VEL
LIN {X 0,Y 467.613,Z 382.36,A -85,B 0,C 180,E1 -7615.109,E2 -7615.109} C_VEL
LIN {X 0,Y 469.105,Z 390.082,A -85,B 0,C 180,E1 -7617.873,E2 -7617.873} C_VEL
LIN {X 0,Y 469.794,Z 394.696,A -85,B 0,C 180,E1 -7619.43,E2 -7619.43} C_VEL
LIN {X 0,Y 469.356,Z 402.233,A -85,B 0,C 180,E1 -7621.781,E2 -7621.781} C_VEL
LIN {X 0,Y 468.676,Z 413.647,A -85,B 0,C 180,E1 -7625.176,E2 -7625.176} C_VEL
LIN {X 0,Y 468.084,Z 425.462,A -85,B 0,C 180,E1 -7628.575,E2 -7628.575} C_VEL
LIN {X 0,Y 467.597,Z 438.009,A -85,B 0,C 180,E1 -7632.057,E2 -7632.057} C_VEL
LIN {X 0,Y 467.318,Z 447.973,A -85,B 0,C 180,E1 -7634.771,E2 -7634.771} C_VEL
LIN {X 0,Y 469.266,Z 463.126,A -85,B 0,C 180,E1 -7635.225,E2 -7635.225} C_VEL
LIN {X 0,Y 469.733,Z 468.524,A -85,B 0,C 180,E1 -7635.433,E2 -7635.433} C_VEL
LIN {X 0,Y 469.253,Z 481.367,A -85,B 0,C 180,E1 -7636.027,E2 -7636.027} C_VEL
LIN {X 0,Y 468.78,Z 493.595,A -85,B 0,C 180,E1 -7636.786,E2 -7636.786} C_VEL
LIN {X 0,Y 468.356,Z 503.581,A -85,B 0,C 180,E1 -7637.576,E2 -7637.576} C_VEL
LIN {X 0,Y 468.024,Z 513.295,A -85,B 0,C 180,E1 -7638.526,E2 -7638.526} C_VEL
LIN {X 0,Y 467.524,Z 522.393,A -85,B 0,C 180,E1 -7639.61,E2 -7639.61} C_VEL
LIN {X 0,Y 467.216,Z 531.27,A -85,B 0,C 180,E1 -7640.915,E2 -7640.915} C_VEL
LIN {X 0,Y 466.958,Z 538.34,A -85,B 0,C 180,E1 -7642.217,E2 -7642.217} C_VEL
LIN {X 0,Y 466.748,Z 544.336,A -85,B 0,C 180,E1 -7643.612,E2 -7643.612} C_VEL
LIN {X 0,Y 466.771,Z 548.415,A -85,B 0,C 180,E1 -7644.819,E2 -7644.819} C_VEL
LIN {X 0,Y 466.664,Z 550.751,A -85,B 0,C 180,E1 -7645.684,E2 -7645.684} C_VEL
LIN {X 0,Y 466.728,Z 552.66,A -85,B 0,C 180,E1 -7646.549,E2 -7646.549} C_VEL
LIN {X 0,Y 466.701,Z 554.094,A -85,B 0,C 180,E1 -7647.413,E2 -7647.413} C_VEL
LIN {X 0,Y 466.693,Z 555.107,A -85,B 0,C 180,E1 -7648.276,E2 -7648.276} C_VEL
LIN {X 0,Y 466.62,Z 555.726,A -85,B 0,C 180,E1 -7649.139,E2 -7649.139} C_VEL
LIN {X 0,Y 466.599,Z 555.944,A -85,B 0,C 180,E1 -7650.002,E2 -7650.002} C_VEL
LIN {X 0,Y 466.694,Z 555.122,A -85,B 0,C 180,E1 -7651.728,E2 -7651.728} C_VEL
LIN {X 0,Y 466.701,Z 554.118,A -85,B 0,C 180,E1 -7652.591,E2 -7652.591} C_VEL
LIN {X 0,Y 466.729,Z 552.699,A -85,B 0,C 180,E1 -7653.455,E2 -7653.455} C_VEL
LIN {X 0,Y 466.698,Z 549.725,A -85,B 0,C 180,E1 -7654.753,E2 -7654.753} C_VEL
LIN {X 0,Y 466.77,Z 545.692,A -85,B 0,C 180,E1 -7656.052,E2 -7656.052} C_VEL
LIN {X 0,Y 466.929,Z 539.461,A -85,B 0,C 180,E1 -7657.57,E2 -7657.57} C_VEL
LIN {X 0,Y 467.156,Z 532.66,A -85,B 0,C 180,E1 -7658.872,E2 -7658.872} C_VEL
LIN {X 0,Y 467.46,Z 524.181,A -85,B 0,C 180,E1 -7660.177,E2 -7660.177} C_VEL
LIN {X 0,Y 467.899,Z 515.427,A -85,B 0,C 180,E1 -7661.262,E2 -7661.262} C_VEL
LIN {X 0,Y 468.285,Z 505.365,A -85,B 0,C 180,E1 -7662.281,E2 -7662.281} C_VEL
LIN {X 0,Y 468.795,Z 493.8,A -85,B 0,C 180,E1 -7663.218,E2 -7663.218} C_VEL
LIN {X 0,Y 469.289,Z 481.608,A -85,B 0,C 180,E1 -7663.976,E2 -7663.976} C_VEL
LIN {X 0,Y 469.726,Z 468.8,A -85,B 0,C 180,E1 -7664.571,E2 -7664.571} C_VEL
LIN {X 0,Y 469.204,Z 462.55,A -85,B 0,C 180,E1 -7664.809,E2 -7664.809} C_VEL
LIN {X 0,Y 467.387,Z 448.881,A -85,B 0,C 180,E1 -7665.202,E2 -7665.202} C_VEL
LIN {X 0,Y 467.319,Z 448.191,A -85,B 0,C 180,E1 -7665.233,E2 -7665.233} C_VEL
LIN {X 0,Y 467.646,Z 436.561,A -85,B 0,C 180,E1 -7668.398,E2 -7668.398} C_VEL
LIN {X 0,Y 468.134,Z 424.736,A -85,B 0,C 180,E1 -7671.682,E2 -7671.682} C_VEL
LIN {X 0,Y 468.695,Z 413.742,A -85,B 0,C 180,E1 -7674.827,E2 -7674.827} C_VEL
LIN {X 0,Y 469.368,Z 402.175,A -85,B 0,C 180,E1 -7678.221,E2 -7678.221} C_VEL
LIN {X 0,Y 469.723,Z 394.454,A -85,B 0,C 180,E1 -7680.579,E2 -7680.579} C_VEL
LIN {X 0,Y 468.712,Z 388.059,A -85,B 0,C 180,E1 -7682.671,E2 -7682.671} C_VEL
LIN {X 0,Y 467.624,Z 382.236,A -85,B 0,C 180,E1 -7684.671,E2 -7684.671} C_VEL
LIN {X 0,Y 467.568,Z 382.246,A -85,B 0,C 180,E1 -7688.046,E2 -7688.046} C_VEL
LIN {X 0,Y 467.566,Z 382.243,A -85,B 0,C 180,E1 -7691.275,E2 -7691.275} C_VEL
LIN {X 0,Y 467.569,Z 382.244,A -85,B 0,C 180,E1 -7695.053,E2 -7695.053} C_VEL
LIN {X 0,Y 467.568,Z 382.243,A -85,B 0,C 180,E1 -7698.726,E2 -7698.726} C_VEL
LIN {X 0,Y 467.57,Z 382.238,A -85,B 0,C 180,E1 -7701.956,E2 -7701.956} C_VEL
LIN {X 0,Y 467.564,Z 382.241,A -85,B 0,C 180,E1 -7705.167,E2 -7705.167} C_VEL
LIN {X 0,Y 467.583,Z 382.241,A -85,B 0,C 180,E1 -7708.26,E2 -7708.26} C_VEL
LIN {X 0,Y 467.548,Z 382.247,A -85,B 0,C 180,E1 -7711.248,E2 -7711.248} C_VEL
LIN {X 0,Y 467.566,Z 382.242,A -85,B 0,C 180,E1 -7714.405,E2 -7714.405} C_VEL
LIN {X 0,Y 467.577,Z 382.244,A -85,B 0,C 180,E1 -7716.996,E2 -7716.996} C_VEL
LIN {X 0,Y 467.628,Z 382.234,A -85,B 0,C 180,E1 -7719.777,E2 -7719.777} C_VEL
LIN {X 0,Y 467.612,Z 382.24,A -85,B 0,C 180,E1 -7722.507,E2 -7722.507} C_VEL
LIN {X 0,Y 467.61,Z 382.238,A -85,B 0,C 180,E1 -7725.196,E2 -7725.196} C_VEL
LIN {X 0,Y 467.66,Z 382.234,A -85,B 0,C 180,E1 -7727.854,E2 -7727.854} C_VEL
LIN {X 0,Y 467.638,Z 382.237,A -85,B 0,C 180,E1 -7731.356,E2 -7731.356} C_VEL
LIN {X 0,Y 467.708,Z 382.225,A -85,B 0,C 180,E1 -7733.962,E2 -7733.962} C_VEL
LIN {X 0,Y 467.535,Z 382.248,A -85,B 0,C 180,E1 -7735.689,E2 -7735.689} C_VEL
LIN {X 0,Y 467.448,Z 382.389,A -85,B 0,C 180,E1 -7736.822,E2 -7736.822} C_VEL
LIN {X 0,Y 467.598,Z 388.908,A -85,B 0,C 180,E1 -7739.569,E2 -7739.569} C_VEL
LIN {X 0,Y 467.299,Z 395.011,A -85,B 0,C 180,E1 -7742.154,E2 -7742.154} C_VEL
LIN {X 0,Y 467.3,Z 401.893,A -85,B 0,C 180,E1 -7745.177,E2 -7745.177} C_VEL
LIN {X 0,Y 467.24,Z 407.767,A -85,B 0,C 180,E1 -7747.78,E2 -7747.78} C_VEL
LIN {X 0,Y 467.132,Z 415.596,A -85,B 0,C 180,E1 -7751.279,E2 -7751.279} C_VEL
LIN {X 0,Y 466.963,Z 423.415,A -85,B 0,C 180,E1 -7754.824,E2 -7754.824} C_VEL
LIN {X 0,Y 466.978,Z 425.506,A -85,B 0,C 180,E1 -7755.684,E2 -7755.684} C_VEL
LIN {X 0,Y 469.739,Z 439.287,A -85,B 0,C 180,E1 -7756.179,E2 -7756.179} C_VEL
LIN {X 0,Y 470.116,Z 444.312,A -85,B 0,C 180,E1 -7756.389,E2 -7756.389} C_VEL
LIN {X 0,Y 469.699,Z 456.243,A -85,B 0,C 180,E1 -7756.959,E2 -7756.959} C_VEL
LIN {X 0,Y 469.25,Z 467.312,A -85,B 0,C 180,E1 -7757.655,E2 -7757.655} C_VEL
LIN {X 0,Y 468.765,Z 478.577,A -85,B 0,C 180,E1 -7758.55,E2 -7758.55} C_VEL
LIN {X 0,Y 468.342,Z 488.277,A -85,B 0,C 180,E1 -7759.505,E2 -7759.505} C_VEL
LIN {X 0,Y 467.887,Z 497.844,A -85,B 0,C 180,E1 -7760.67,E2 -7760.67} C_VEL
LIN {X 0,Y 467.491,Z 505.794,A -85,B 0,C 180,E1 -7761.859,E2 -7761.859} C_VEL
LIN {X 0,Y 467.244,Z 512.162,A -85,B 0,C 180,E1 -7763.021,E2 -7763.021} C_VEL
LIN {X 0,Y 466.891,Z 518.487,A -85,B 0,C 180,E1 -7764.453,E2 -7764.453} C_VEL
LIN {X 0,Y 466.79,Z 523.286,A -85,B 0,C 180,E1 -7765.888,E2 -7765.888} C_VEL
LIN {X 0,Y 466.673,Z 526.77,A -85,B 0,C 180,E1 -7767.31,E2 -7767.31} C_VEL
LIN {X 0,Y 466.541,Z 529.529,A -85,B 0,C 180,E1 -7769.105,E2 -7769.105} C_VEL
LIN {X 0,Y 466.529,Z 530.492,A -85,B 0,C 180,E1 -7770.81,E2 -7770.81} C_VEL
LIN {X 0,Y 466.524,Z 529.958,A -85,B 0,C 180,E1 -7772.475,E2 -7772.475} C_VEL
LIN {X 0,Y 466.577,Z 528.026,A -85,B 0,C 180,E1 -7774.058,E2 -7774.058} C_VEL
LIN {X 0,Y 466.72,Z 524.83,A -85,B 0,C 180,E1 -7775.594,E2 -7775.594} C_VEL
LIN {X 0,Y 466.902,Z 520.375,A -85,B 0,C 180,E1 -7777.08,E2 -7777.08} C_VEL
LIN {X 0,Y 467.087,Z 514.61,A -85,B 0,C 180,E1 -7778.516,E2 -7778.516} C_VEL
LIN {X 0,Y 467.383,Z 507.413,A -85,B 0,C 180,E1 -7779.924,E2 -7779.924} C_VEL
LIN {X 0,Y 467.7,Z 500.174,A -85,B 0,C 180,E1 -7781.066,E2 -7781.066} C_VEL
LIN {X 0,Y 468.11,Z 491.296,A -85,B 0,C 180,E1 -7782.21,E2 -7782.21} C_VEL
LIN {X 0,Y 468.651,Z 480.383,A -85,B 0,C 180,E1 -7783.347,E2 -7783.347} C_VEL
LIN {X 0,Y 469.065,Z 470.036,A -85,B 0,C 180,E1 -7784.213,E2 -7784.213} C_VEL
LIN {X 0,Y 469.537,Z 457.746,A -85,B 0,C 180,E1 -7785.019,E2 -7785.019} C_VEL
LIN {X 0,Y 470.07,Z 444.825,A -85,B 0,C 180,E1 -7785.656,E2 -7785.656} C_VEL
LIN {X 0,Y 469.624,Z 438.866,A -85,B 0,C 180,E1 -7785.902,E2 -7785.902} C_VEL
LIN {X 0,Y 466.91,Z 424.905,A -85,B 0,C 180,E1 -7786.401,E2 -7786.401} C_VEL
LIN {X 0,Y 467.017,Z 417.824,A -85,B 0,C 180,E1 -7789.676,E2 -7789.676} C_VEL
LIN {X 0,Y 467.077,Z 410.883,A -85,B 0,C 180,E1 -7792.889,E2 -7792.889} C_VEL
LIN {X 0,Y 467.289,Z 404.553,A -85,B 0,C 180,E1 -7795.811,E2 -7795.811} C_VEL
LIN {X 0,Y 467.39,Z 397.117,A -85,B 0,C 180,E1 -7799.252,E2 -7799.252} C_VEL
LIN {X 0,Y 467.414,Z 390.044,A -85,B 0,C 180,E1 -7802.513,E2 -7802.513} C_VEL
LIN {X 0,Y 467.414,Z 389.278,A -85,B 0,C 180,E1 -7802.87,E2 -7802.87} C_VEL
LIN {X 0,Y 466.794,Z 387.873,A -85,B 0,C 180,E1 -7803.566,E2 -7803.566} C_VEL
LIN {X 0,Y 464.071,Z 385.711,A -85,B 0,C 180,E1 -7804.703,E2 -7804.703} C_VEL
LIN {X 0,Y 461.725,Z 384.031,A -85,B 0,C 180,E1 -7805.627,E2 -7805.627} C_VEL
LIN {X 0,Y 460.673,Z 383.188,A -85,B 0,C 180,E1 -7806.348,E2 -7806.348} C_VEL
LIN {X 0,Y 460.564,Z 383.117,A -85,B 0,C 180,E1 -7806.594,E2 -7806.594} C_VEL
LIN {X 0,Y 460.553,Z 383.116,A -85,B 0,C 180,E1 -7809.451,E2 -7809.451} C_VEL
LIN {X 0,Y 460.549,Z 383.119,A -85,B 0,C 180,E1 -7812.228,E2 -7812.228} C_VEL
LIN {X 0,Y 460.567,Z 383.117,A -85,B 0,C 180,E1 -7814.963,E2 -7814.963} C_VEL
LIN {X 0,Y 460.61,Z 383.111,A -85,B 0,C 180,E1 -7818.558,E2 -7818.558} C_VEL
LIN {X 0,Y 460.667,Z 383.102,A -85,B 0,C 180,E1 -7822.106,E2 -7822.106} C_VEL
LIN {X 0,Y 460.687,Z 383.105,A -85,B 0,C 180,E1 -7824.746,E2 -7824.746} C_VEL
LIN {X 0,Y 460.758,Z 383.093,A -85,B 0,C 180,E1 -7827.375,E2 -7827.375} C_VEL
LIN {X 0,Y 460.854,Z 383.284,A -85,B 0,C 180,E1 -7829.78,E2 -7829.78} C_VEL
LIN {X 0,Y 460.702,Z 386.775,A -85,B 0,C 180,E1 -7831.746,E2 -7831.746} C_VEL
LIN {X 0,Y 460.584,Z 393.038,A -85,B 0,C 180,E1 -7835.251,E2 -7835.251} C_VEL
LIN {X 0,Y 460.315,Z 399.493,A -85,B 0,C 180,E1 -7838.78,E2 -7838.78} C_VEL
LIN {X 0,Y 460.152,Z 406.084,A -85,B 0,C 180,E1 -7842.344,E2 -7842.344} C_VEL
LIN {X 0,Y 459.92,Z 412.917,A -85,B 0,C 180,E1 -7845.963,E2 -7845.963} C_VEL
LIN {X 0,Y 459.788,Z 418.19,A -85,B 0,C 180,E1 -7848.72,E2 -7848.72} C_VEL
LIN {X 0,Y 459.793,Z 421.656,A -85,B 0,C 180,E1 -7850.522,E2 -7850.522} C_VEL
LIN {X 0,Y 461.91,Z 433.448,A -85,B 0,C 180,E1 -7851.005,E2 -7851.005} C_VEL
LIN {X 0,Y 462.243,Z 438.389,A -85,B 0,C 180,E1 -7851.244,E2 -7851.244} C_VEL
LIN {X 0,Y 461.808,Z 449.408,A -85,B 0,C 180,E1 -7851.88,E2 -7851.88} C_VEL
LIN {X 0,Y 461.379,Z 459.039,A -85,B 0,C 180,E1 -7852.618,E2 -7852.618} C_VEL
LIN {X 0,Y 461.061,Z 468.074,A -85,B 0,C 180,E1 -7853.494,E2 -7853.494} C_VEL
LIN {X 0,Y 460.7,Z 476.744,A -85,B 0,C 180,E1 -7854.561,E2 -7854.561} C_VEL
LIN {X 0,Y 460.319,Z 484.298,A -85,B 0,C 180,E1 -7855.738,E2 -7855.738} C_VEL
LIN {X 0,Y 460.01,Z 490.759,A -85,B 0,C 180,E1 -7857.031,E2 -7857.031} C_VEL
LIN {X 0,Y 459.835,Z 495.468,A -85,B 0,C 180,E1 -7858.278,E2 -7858.278} C_VEL
LIN {X 0,Y 459.789,Z 498.642,A -85,B 0,C 180,E1 -7859.395,E2 -7859.395} C_VEL
LIN {X 0,Y 459.655,Z 500.569,A -85,B 0,C 180,E1 -7860.299,E2 -7860.299} C_VEL
LIN {X 0,Y 459.543,Z 502.08,A -85,B 0,C 180,E1 -7861.328,E2 -7861.328} C_VEL
LIN {X 0,Y 459.51,Z 502.999,A -85,B 0,C 180,E1 -7862.733,E2 -7862.733} C_VEL
LIN {X 0,Y 459.531,Z 503.003,A -85,B 0,C 180,E1 -7863.403,E2 -7863.403} C_VEL
LIN {X 0,Y 459.579,Z 502.427,A -85,B 0,C 180,E1 -7864.455,E2 -7864.455} C_VEL
LIN {X 0,Y 459.678,Z 500.538,A -85,B 0,C 180,E1 -7865.874,E2 -7865.874} C_VEL
LIN {X 0,Y 459.883,Z 496.993,A -85,B 0,C 180,E1 -7867.376,E2 -7867.376} C_VEL
LIN {X 0,Y 460.066,Z 491.965,A -85,B 0,C 180,E1 -7868.824,E2 -7868.824} C_VEL
LIN {X 0,Y 460.255,Z 487.109,A -85,B 0,C 180,E1 -7869.887,E2 -7869.887} C_VEL
LIN {X 0,Y 460.538,Z 480.724,A -85,B 0,C 180,E1 -7871.007,E2 -7871.007} C_VEL
LIN {X 0,Y 460.882,Z 472.532,A -85,B 0,C 180,E1 -7872.137,E2 -7872.137} C_VEL
LIN {X 0,Y 461.339,Z 463.936,A -85,B 0,C 180,E1 -7873.078,E2 -7873.078} C_VEL
LIN {X 0,Y 461.787,Z 453.508,A -85,B 0,C 180,E1 -7873.973,E2 -7873.973} C_VEL
LIN {X 0,Y 462.177,Z 442.084,A -85,B 0,C 180,E1 -7874.709,E2 -7874.709} C_VEL
LIN {X 0,Y 462.24,Z 435.049,A -85,B 0,C 180,E1 -7875.061,E2 -7875.061} C_VEL
LIN {X 0,Y 460.077,Z 423.454,A -85,B 0,C 180,E1 -7875.561,E2 -7875.561} C_VEL
LIN {X 0,Y 459.806,Z 421.958,A -85,B 0,C 180,E1 -7875.641,E2 -7875.641} C_VEL
LIN {X 0,Y 459.889,Z 416.577,A -85,B 0,C 180,E1 -7878.483,E2 -7878.483} C_VEL
LIN {X 0,Y 460.021,Z 410.389,A -85,B 0,C 180,E1 -7881.776,E2 -7881.776} C_VEL
LIN {X 0,Y 460.132,Z 405.33,A -85,B 0,C 180,E1 -7884.521,E2 -7884.521} C_VEL
LIN {X 0,Y 460.323,Z 399.476,A -85,B 0,C 180,E1 -7887.7,E2 -7887.7} C_VEL
LIN {X 0,Y 460.48,Z 393.921,A -85,B 0,C 180,E1 -7890.765,E2 -7890.765} C_VEL
LIN {X 0,Y 460.742,Z 387.907,A -85,B 0,C 180,E1 -7894.146,E2 -7894.146} C_VEL
LIN {X 0,Y 460.662,Z 383.566,A -85,B 0,C 180,E1 -7896.631,E2 -7896.631} C_VEL
LIN {X 0,Y 460.576,Z 383.119,A -85,B 0,C 180,E1 -7897.101,E2 -7897.101} C_VEL
LIN {X 0,Y 460.546,Z 383.122,A -85,B 0,C 180,E1 -7900.384,E2 -7900.384} C_VEL
LIN {X 0,Y 460.541,Z 383.124,A -85,B 0,C 180,E1 -7903.146,E2 -7903.146} C_VEL
LIN {X 0,Y 460.541,Z 383.121,A -85,B 0,C 180,E1 -7905.868,E2 -7905.868} C_VEL
LIN {X 0,Y 460.617,Z 383.111,A -85,B 0,C 180,E1 -7908.56,E2 -7908.56} C_VEL
LIN {X 0,Y 460.671,Z 383.102,A -85,B 0,C 180,E1 -7912.108,E2 -7912.108} C_VEL
LIN {X 0,Y 460.684,Z 383.101,A -85,B 0,C 180,E1 -7914.748,E2 -7914.748} C_VEL
LIN {X 0,Y 460.811,Z 383.085,A -85,B 0,C 180,E1 -7917.378,E2 -7917.378} C_VEL
LIN {X 0,Y 460.828,Z 383.083,A -85,B 0,C 180,E1 -7920,E2 -7920} C_VEL
LIN {X 0,Y 460.811,Z 383.085,A -85,B 0,C 180,E1 -7922.623,E2 -7922.623} C_VEL
LIN {X 0,Y 460.696,Z 383.098,A -85,B 0,C 180,E1 -7926.13,E2 -7926.13} C_VEL
LIN {X 0,Y 460.608,Z 383.11,A -85,B 0,C 180,E1 -7928.777,E2 -7928.777} C_VEL
LIN {X 0,Y 460.627,Z 383.107,A -85,B 0,C 180,E1 -7932.467,E2 -7932.467} C_VEL
LIN {X 0,Y 460.598,Z 383.109,A -85,B 0,C 180,E1 -7936.008,E2 -7936.008} C_VEL
LIN {X 0,Y 460.553,Z 383.114,A -85,B 0,C 180,E1 -7938.905,E2 -7938.905} C_VEL
LIN {X 0,Y 460.542,Z 383.116,A -85,B 0,C 180,E1 -7941.485,E2 -7941.485} C_VEL
LIN {X 0,Y 460.524,Z 383.119,A -85,B 0,C 180,E1 -7944.334,E2 -7944.334} C_VEL
LIN {X 0,Y 460.563,Z 383.115,A -85,B 0,C 180,E1 -7947.245,E2 -7947.245} C_VEL
LIN {X 0,Y 460.507,Z 383.123,A -85,B 0,C 180,E1 -7950.241,E2 -7950.241} C_VEL
LIN {X 0,Y 460.511,Z 383.122,A -85,B 0,C 180,E1 -7953.327,E2 -7953.327} C_VEL
LIN {X 0,Y 460.462,Z 383.13,A -85,B 0,C 180,E1 -7956.531,E2 -7956.531} C_VEL
LIN {X 0,Y 460.562,Z 383.116,A -85,B 0,C 180,E1 -7959.86,E2 -7959.86} C_VEL
LIN {X 0,Y 460.527,Z 383.121,A -85,B 0,C 180,E1 -7962.907,E2 -7962.907} C_VEL
LIN {X 0,Y 460.51,Z 383.123,A -85,B 0,C 180,E1 -7965.831,E2 -7965.831} C_VEL
LIN {X 0,Y 460.53,Z 383.123,A -85,B 0,C 180,E1 -7968.992,E2 -7968.992} C_VEL
LIN {X 0,Y 460.536,Z 383.121,A -85,B 0,C 180,E1 -7971.272,E2 -7971.272} C_VEL
LIN {X 0,Y 460.574,Z 383.312,A -85,B 0,C 180,E1 -7974.801,E2 -7974.801} C_VEL
LIN {X 0,Y 462.186,Z 391.66,A -85,B 0,C 180,E1 -7977.848,E2 -7977.848} C_VEL
LIN {X 0,Y 462.865,Z 396.255,A -85,B 0,C 180,E1 -7979.429,E2 -7979.429} C_VEL
LIN {X 0,Y 462.343,Z 404.01,A -85,B 0,C 180,E1 -7981.889,E2 -7981.889} C_VEL
LIN {X 0,Y 461.648,Z 415.161,A -85,B 0,C 180,E1 -7985.253,E2 -7985.253} C_VEL
LIN {X 0,Y 461.04,Z 426.347,A -85,B 0,C 180,E1 -7988.543,E2 -7988.543} C_VEL
LIN {X 0,Y 460.559,Z 437.75,A -85,B 0,C 180,E1 -7991.773,E2 -7991.773} C_VEL
LIN {X 0,Y 460.24,Z 447.78,A -85,B 0,C 180,E1 -7994.566,E2 -7994.566} C_VEL
LIN {X 0,Y 462.113,Z 461.926,A -85,B 0,C 180,E1 -7994.98,E2 -7994.98} C_VEL
LIN {X 0,Y 462.799,Z 469.118,A -85,B 0,C 180,E1 -7995.267,E2 -7995.267} C_VEL
LIN {X 0,Y 462.293,Z 481.738,A -85,B 0,C 180,E1 -7995.868,E2 -7995.868} C_VEL
LIN {X 0,Y 461.839,Z 493.03,A -85,B 0,C 180,E1 -7996.584,E2 -7996.584} C_VEL
LIN {X 0,Y 461.352,Z 503.598,A -85,B 0,C 180,E1 -7997.434,E2 -7997.434} C_VEL
LIN {X 0,Y 461.031,Z 512.817,A -85,B 0,C 180,E1 -7998.349,E2 -7998.349} C_VEL
LIN {X 0,Y 460.5,Z 521.933,A -85,B 0,C 180,E1 -7999.45,E2 -7999.45} C_VEL
LIN {X 0,Y 460.176,Z 530.825,A -85,B 0,C 180,E1 -8000.774,E2 -8000.774} C_VEL
LIN {X 0,Y 459.889,Z 537.914,A -85,B 0,C 180,E1 -8002.097,E2 -8002.097} C_VEL
LIN {X 0,Y 459.673,Z 544.294,A -85,B 0,C 180,E1 -8003.615,E2 -8003.615} C_VEL
LIN {X 0,Y 459.627,Z 549.249,A -85,B 0,C 180,E1 -8005.178,E2 -8005.178} C_VEL
LIN {X 0,Y 459.625,Z 552.248,A -85,B 0,C 180,E1 -8006.495,E2 -8006.495} C_VEL
LIN {X 0,Y 459.621,Z 553.693,A -85,B 0,C 180,E1 -8007.373,E2 -8007.373} C_VEL
LIN {X 0,Y 459.614,Z 554.712,A -85,B 0,C 180,E1 -8008.249,E2 -8008.249} C_VEL
LIN {X 0,Y 459.553,Z 555.328,A -85,B 0,C 180,E1 -8009.126,E2 -8009.126} C_VEL
LIN {X 0,Y 459.53,Z 555.541,A -85,B 0,C 180,E1 -8010.002,E2 -8010.002} C_VEL
LIN {X 0,Y 459.63,Z 554.719,A -85,B 0,C 180,E1 -8011.754,E2 -8011.754} C_VEL
LIN {X 0,Y 459.622,Z 553.714,A -85,B 0,C 180,E1 -8012.631,E2 -8012.631} C_VEL
LIN {X 0,Y 459.626,Z 552.29,A -85,B 0,C 180,E1 -8013.508,E2 -8013.508} C_VEL
LIN {X 0,Y 459.629,Z 549.314,A -85,B 0,C 180,E1 -8014.826,E2 -8014.826} C_VEL
LIN {X 0,Y 459.716,Z 544.217,A -85,B 0,C 180,E1 -8016.433,E2 -8016.433} C_VEL
LIN {X 0,Y 459.893,Z 538.018,A -85,B 0,C 180,E1 -8017.907,E2 -8017.907} C_VEL
LIN {X 0,Y 460.181,Z 530.947,A -85,B 0,C 180,E1 -8019.229,E2 -8019.229} C_VEL
LIN {X 0,Y 460.502,Z 522.072,A -85,B 0,C 180,E1 -8020.554,E2 -8020.554} C_VEL
LIN {X 0,Y 461.048,Z 512.972,A -85,B 0,C 180,E1 -8021.654,E2 -8021.654} C_VEL
LIN {X 0,Y 461.369,Z 503.709,A -85,B 0,C 180,E1 -8022.575,E2 -8022.575} C_VEL
LIN {X 0,Y 461.834,Z 493.19,A -85,B 0,C 180,E1 -8023.421,E2 -8023.421} C_VEL
LIN {X 0,Y 462.394,Z 480.918,A -85,B 0,C 180,E1 -8024.189,E2 -8024.189} C_VEL
LIN {X 0,Y 462.822,Z 467.936,A -85,B 0,C 180,E1 -8024.793,E2 -8024.793} C_VEL
LIN {X 0,Y 461.243,Z 454.822,A -85,B 0,C 180,E1 -8025.255,E2 -8025.255} C_VEL
LIN {X 0,Y 460.275,Z 447.971,A -85,B 0,C 180,E1 -8025.444,E2 -8025.444} C_VEL
LIN {X 0,Y 460.678,Z 435.406,A -85,B 0,C 180,E1 -8028.939,E2 -8028.939} C_VEL
LIN {X 0,Y 461.21,Z 423.292,A -85,B 0,C 180,E1 -8032.394,E2 -8032.394} C_VEL
LIN {X 0,Y 461.833,Z 412.003,A -85,B 0,C 180,E1 -8035.684,E2 -8035.684} C_VEL
LIN {X 0,Y 462.573,Z 400.733,A -85,B 0,C 180,E1 -8039.092,E2 -8039.092} C_VEL
LIN {X 0,Y 462.78,Z 395.941,A -85,B 0,C 180,E1 -8040.582,E2 -8040.582} C_VEL
LIN {X 0,Y 461.82,Z 389.748,A -85,B 0,C 180,E1 -8042.647,E2 -8042.647} C_VEL
LIN {X 0,Y 460.573,Z 383.117,A -85,B 0,C 180,E1 -8045.01,E2 -8045.01} C_VEL
LIN {X 0,Y 460.52,Z 383.122,A -85,B 0,C 180,E1 -8048.735,E2 -8048.735} C_VEL
LIN {X 0,Y 460.508,Z 383.125,A -85,B 0,C 180,E1 -8051.599,E2 -8051.599} C_VEL
LIN {X 0,Y 460.512,Z 383.12,A -85,B 0,C 180,E1 -8054.59,E2 -8054.59} C_VEL
LIN {X 0,Y 460.485,Z 383.123,A -85,B 0,C 180,E1 -8057.814,E2 -8057.814} C_VEL
LIN {X 0,Y 460.519,Z 383.118,A -85,B 0,C 180,E1 -8060.136,E2 -8060.136} C_VEL
LIN {X 0,Y 460.482,Z 383.123,A -85,B 0,C 180,E1 -8063.471,E2 -8063.471} C_VEL
LIN {X 0,Y 460.523,Z 383.119,A -85,B 0,C 180,E1 -8066.674,E2 -8066.674} C_VEL
LIN {X 0,Y 460.509,Z 383.125,A -85,B 0,C 180,E1 -8069.76,E2 -8069.76} C_VEL
LIN {X 0,Y 460.489,Z 383.124,A -85,B 0,C 180,E1 -8072.751,E2 -8072.751} C_VEL
LIN {X 0,Y 460.517,Z 383.12,A -85,B 0,C 180,E1 -8075.666,E2 -8075.666} C_VEL
LIN {X 0,Y 460.527,Z 383.123,A -85,B 0,C 180,E1 -8078.578,E2 -8078.578} C_VEL
LIN {X 0,Y 460.596,Z 383.11,A -85,B 0,C 180,E1 -8081.311,E2 -8081.311} C_VEL
LIN {X 0,Y 460.61,Z 383.114,A -85,B 0,C 180,E1 -8084.059,E2 -8084.059} C_VEL
LIN {X 0,Y 460.614,Z 383.112,A -85,B 0,C 180,E1 -8087.666,E2 -8087.666} C_VEL
LIN {X 0,Y 460.593,Z 383.115,A -85,B 0,C 180,E1 -8091.223,E2 -8091.223} C_VEL
LIN {X 0,Y 460.674,Z 383.102,A -85,B 0,C 180,E1 -8093.869,E2 -8093.869} C_VEL
LIN {X 0,Y 460.498,Z 383.125,A -85,B 0,C 180,E1 -8095.623,E2 -8095.623} C_VEL
LIN {X 0,Y 460.404,Z 383.237,A -85,B 0,C 180,E1 -8096.718,E2 -8096.718} C_VEL
LIN {X 0,Y 460.57,Z 389.935,A -85,B 0,C 180,E1 -8099.563,E2 -8099.563} C_VEL
LIN {X 0,Y 460.255,Z 396.052,A -85,B 0,C 180,E1 -8102.187,E2 -8102.187} C_VEL
LIN {X 0,Y 460.257,Z 402.884,A -85,B 0,C 180,E1 -8105.256,E2 -8105.256} C_VEL
LIN {X 0,Y 460.183,Z 408.93,A -85,B 0,C 180,E1 -8107.9,E2 -8107.9} C_VEL
LIN {X 0,Y 460.071,Z 416.785,A -85,B 0,C 180,E1 -8111.454,E2 -8111.454} C_VEL
LIN {X 0,Y 459.917,Z 424.653,A -85,B 0,C 180,E1 -8115.057,E2 -8115.057} C_VEL
LIN {X 0,Y 459.95,Z 425.7,A -85,B 0,C 180,E1 -8115.435,E2 -8115.435} C_VEL
LIN {X 0,Y 462.72,Z 439.279,A -85,B 0,C 180,E1 -8115.935,E2 -8115.935} C_VEL
LIN {X 0,Y 463.27,Z 444.493,A -85,B 0,C 180,E1 -8116.161,E2 -8116.161} C_VEL
LIN {X 0,Y 462.804,Z 456.948,A -85,B 0,C 180,E1 -8116.77,E2 -8116.77} C_VEL
LIN {X 0,Y 462.296,Z 469.426,A -85,B 0,C 180,E1 -8117.587,E2 -8117.587} C_VEL
LIN {X 0,Y 461.744,Z 480.628,A -85,B 0,C 180,E1 -8118.525,E2 -8118.525} C_VEL
LIN {X 0,Y 461.235,Z 490.726,A -85,B 0,C 180,E1 -8119.586,E2 -8119.586} C_VEL
LIN {X 0,Y 460.768,Z 499.905,A -85,B 0,C 180,E1 -8120.77,E2 -8120.77} C_VEL
LIN {X 0,Y 460.41,Z 507.423,A -85,B 0,C 180,E1 -8121.961,E2 -8121.961} C_VEL
LIN {X 0,Y 460.044,Z 514.721,A -85,B 0,C 180,E1 -8123.403,E2 -8123.403} C_VEL
LIN {X 0,Y 459.821,Z 520.486,A -85,B 0,C 180,E1 -8124.854,E2 -8124.854} C_VEL
LIN {X 0,Y 459.668,Z 524.875,A -85,B 0,C 180,E1 -8126.32,E2 -8126.32} C_VEL
LIN {X 0,Y 459.563,Z 527.465,A -85,B 0,C 180,E1 -8127.502,E2 -8127.502} C_VEL
LIN {X 0,Y 459.49,Z 528.793,A -85,B 0,C 180,E1 -8128.304,E2 -8128.304} C_VEL
LIN {X 0,Y 459.45,Z 529.939,A -85,B 0,C 180,E1 -8129.318,E2 -8129.318} C_VEL
LIN {X 0,Y 459.42,Z 530.589,A -85,B 0,C 180,E1 -8130.319,E2 -8130.319} C_VEL
LIN {X 0,Y 459.412,Z 530.667,A -85,B 0,C 180,E1 -8131.34,E2 -8131.34} C_VEL
LIN {X 0,Y 459.429,Z 529.944,A -85,B 0,C 180,E1 -8132.716,E2 -8132.716} C_VEL
LIN {X 0,Y 459.516,Z 527.607,A -85,B 0,C 180,E1 -8134.464,E2 -8134.464} C_VEL
LIN {X 0,Y 459.693,Z 523.558,A -85,B 0,C 180,E1 -8136.201,E2 -8136.201} C_VEL
LIN {X 0,Y 459.904,Z 518.693,A -85,B 0,C 180,E1 -8137.68,E2 -8137.68} C_VEL
LIN {X 0,Y 460.121,Z 512.808,A -85,B 0,C 180,E1 -8139.054,E2 -8139.054} C_VEL
LIN {X 0,Y 460.434,Z 505.753,A -85,B 0,C 180,E1 -8140.364,E2 -8140.364} C_VEL
LIN {X 0,Y 460.837,Z 497.231,A -85,B 0,C 180,E1 -8141.644,E2 -8141.644} C_VEL
LIN {X 0,Y 461.288,Z 488.745,A -85,B 0,C 180,E1 -8142.686,E2 -8142.686} C_VEL
LIN {X 0,Y 461.751,Z 478.888,A -85,B 0,C 180,E1 -8143.679,E2 -8143.679} C_VEL
LIN {X 0,Y 462.23,Z 468.439,A -85,B 0,C 180,E1 -8144.532,E2 -8144.532} C_VEL
LIN {X 0,Y 462.729,Z 456.3,A -85,B 0,C 180,E1 -8145.316,E2 -8145.316} C_VEL
LIN {X 0,Y 463.209,Z 444.507,A -85,B 0,C 180,E1 -8145.887,E2 -8145.887} C_VEL
LIN {X 0,Y 462.256,Z 437.057,A -85,B 0,C 180,E1 -8146.204,E2 -8146.204} C_VEL
LIN {X 0,Y 459.876,Z 425.033,A -85,B 0,C 180,E1 -8146.638,E2 -8146.638} C_VEL
LIN {X 0,Y 459.955,Z 417.662,A -85,B 0,C 180,E1 -8150.076,E2 -8150.076} C_VEL
LIN {X 0,Y 460.047,Z 412.241,A -85,B 0,C 180,E1 -8152.597,E2 -8152.597} C_VEL
LIN {X 0,Y 460.229,Z 404.677,A -85,B 0,C 180,E1 -8156.124,E2 -8156.124} C_VEL
LIN {X 0,Y 460.345,Z 397.94,A -85,B 0,C 180,E1 -8159.256,E2 -8159.256} C_VEL
LIN {X 0,Y 460.37,Z 391.385,A -85,B 0,C 180,E1 -8162.303,E2 -8162.303} C_VEL
LIN {X 0,Y 460.575,Z 384.097,A -85,B 0,C 180,E1 -8165.668,E2 -8165.668} C_VEL
LIN {X 0,Y 460.638,Z 383.109,A -85,B 0,C 180,E1 -8166.203,E2 -8166.203} C_VEL
LIN {X 0,Y 460.564,Z 383.117,A -85,B 0,C 180,E1 -8166.594,E2 -8166.594} C_VEL
LIN {X 0,Y 459.837,Z 383.209,A -85,B 0,C 180,E1 -8167.325,E2 -8167.325} C_VEL
LIN {X 0,Y 456.969,Z 383.565,A -85,B 0,C 180,E1 -8168.511,E2 -8168.511} C_VEL
LIN {X 0,Y 454.586,Z 383.86,A -85,B 0,C 180,E1 -8169.467,E2 -8169.467} C_VEL
LIN {X 0,Y 453.576,Z 383.988,A -85,B 0,C 180,E1 -8170.206,E2 -8170.206} C_VEL
LIN {X 0,Y 453.497,Z 383.994,A -85,B 0,C 180,E1 -8170.456,E2 -8170.456} C_VEL
LIN {X 0,Y 453.571,Z 383.987,A -85,B 0,C 180,E1 -8173.878,E2 -8173.878} C_VEL
LIN {X 0,Y 453.565,Z 383.986,A -85,B 0,C 180,E1 -8177.469,E2 -8177.469} C_VEL
LIN {X 0,Y 453.591,Z 383.985,A -85,B 0,C 180,E1 -8181.085,E2 -8181.085} C_VEL
LIN {X 0,Y 453.651,Z 383.978,A -85,B 0,C 180,E1 -8183.773,E2 -8183.773} C_VEL
LIN {X 0,Y 453.705,Z 383.971,A -85,B 0,C 180,E1 -8187.335,E2 -8187.335} C_VEL
LIN {X 0,Y 453.827,Z 384.125,A -85,B 0,C 180,E1 -8189.665,E2 -8189.665} C_VEL
LIN {X 0,Y 453.669,Z 387.788,A -85,B 0,C 180,E1 -8191.773,E2 -8191.773} C_VEL
LIN {X 0,Y 453.532,Z 394.111,A -85,B 0,C 180,E1 -8195.333,E2 -8195.333} C_VEL
LIN {X 0,Y 453.308,Z 398.968,A -85,B 0,C 180,E1 -8198.019,E2 -8198.019} C_VEL
LIN {X 0,Y 453.15,Z 405.559,A -85,B 0,C 180,E1 -8201.629,E2 -8201.629} C_VEL
LIN {X 0,Y 452.901,Z 412.363,A -85,B 0,C 180,E1 -8205.293,E2 -8205.293} C_VEL
LIN {X 0,Y 452.72,Z 418.885,A -85,B 0,C 180,E1 -8208.746,E2 -8208.746} C_VEL
LIN {X 0,Y 452.711,Z 422.027,A -85,B 0,C 180,E1 -8210.323,E2 -8210.323} C_VEL
LIN {X 0,Y 454.724,Z 432.866,A -85,B 0,C 180,E1 -8210.761,E2 -8210.761} C_VEL
LIN {X 0,Y 455.353,Z 438.168,A -85,B 0,C 180,E1 -8211.027,E2 -8211.027} C_VEL
LIN {X 0,Y 454.916,Z 448.88,A -85,B 0,C 180,E1 -8211.642,E2 -8211.642} C_VEL
LIN {X 0,Y 454.432,Z 459.083,A -85,B 0,C 180,E1 -8212.424,E2 -8212.424} C_VEL
LIN {X 0,Y 454.082,Z 468.618,A -85,B 0,C 180,E1 -8213.364,E2 -8213.364} C_VEL
LIN {X 0,Y 453.653,Z 477.784,A -85,B 0,C 180,E1 -8214.518,E2 -8214.518} C_VEL
LIN {X 0,Y 453.29,Z 485.247,A -85,B 0,C 180,E1 -8215.727,E2 -8215.727} C_VEL
LIN {X 0,Y 452.95,Z 491.354,A -85,B 0,C 180,E1 -8216.988,E2 -8216.988} C_VEL
LIN {X 0,Y 452.788,Z 496.013,A -85,B 0,C 180,E1 -8218.252,E2 -8218.252} C_VEL
LIN {X 0,Y 452.689,Z 499.686,A -85,B 0,C 180,E1 -8219.612,E2 -8219.612} C_VEL
LIN {X 0,Y 452.469,Z 502.499,A -85,B 0,C 180,E1 -8221.319,E2 -8221.319} C_VEL
LIN {X 0,Y 452.43,Z 503.455,A -85,B 0,C 180,E1 -8222.984,E2 -8222.984} C_VEL
LIN {X 0,Y 452.499,Z 502.734,A -85,B 0,C 180,E1 -8224.597,E2 -8224.597} C_VEL
LIN {X 0,Y 452.623,Z 500.496,A -85,B 0,C 180,E1 -8226.156,E2 -8226.156} C_VEL
LIN {X 0,Y 452.849,Z 496.758,A -85,B 0,C 180,E1 -8227.675,E2 -8227.675} C_VEL
LIN {X 0,Y 453.08,Z 491.491,A -85,B 0,C 180,E1 -8229.143,E2 -8229.143} C_VEL
LIN {X 0,Y 453.335,Z 485.987,A -85,B 0,C 180,E1 -8230.301,E2 -8230.301} C_VEL
LIN {X 0,Y 453.64,Z 478.964,A -85,B 0,C 180,E1 -8231.472,E2 -8231.472} C_VEL
LIN {X 0,Y 454.022,Z 470.986,A -85,B 0,C 180,E1 -8232.528,E2 -8232.528} C_VEL
LIN {X 0,Y 454.519,Z 460.966,A -85,B 0,C 180,E1 -8233.571,E2 -8233.571} C_VEL
LIN {X 0,Y 455.032,Z 450.042,A -85,B 0,C 180,E1 -8234.438,E2 -8234.438} C_VEL
LIN {X 0,Y 455.384,Z 439.295,A -85,B 0,C 180,E1 -8235.077,E2 -8235.077} C_VEL
LIN {X 0,Y 455.213,Z 435.312,A -85,B 0,C 180,E1 -8235.277,E2 -8235.277} C_VEL
LIN {X 0,Y 453.11,Z 424.091,A -85,B 0,C 180,E1 -8235.774,E2 -8235.774} C_VEL
LIN {X 0,Y 452.748,Z 422.235,A -85,B 0,C 180,E1 -8235.844,E2 -8235.844} C_VEL
LIN {X 0,Y 452.832,Z 416.814,A -85,B 0,C 180,E1 -8238.742,E2 -8238.742} C_VEL
LIN {X 0,Y 452.959,Z 411.453,A -85,B 0,C 180,E1 -8241.638,E2 -8241.638} C_VEL
LIN {X 0,Y 453.095,Z 405.33,A -85,B 0,C 180,E1 -8244.977,E2 -8244.977} C_VEL
LIN {X 0,Y 453.31,Z 399.566,A -85,B 0,C 180,E1 -8248.189,E2 -8248.189} C_VEL
LIN {X 0,Y 453.465,Z 394.013,A -85,B 0,C 180,E1 -8251.285,E2 -8251.285} C_VEL
LIN {X 0,Y 453.724,Z 388.719,A -85,B 0,C 180,E1 -8254.297,E2 -8254.297} C_VEL
LIN {X 0,Y 453.577,Z 384.162,A -85,B 0,C 180,E1 -8256.969,E2 -8256.969} C_VEL
LIN {X 0,Y 453.489,Z 383.999,A -85,B 0,C 180,E1 -8260.066,E2 -8260.066} C_VEL
LIN {X 0,Y 453.482,Z 384.002,A -85,B 0,C 180,E1 -8262.875,E2 -8262.875} C_VEL
LIN {X 0,Y 453.496,Z 383.999,A -85,B 0,C 180,E1 -8265.644,E2 -8265.644} C_VEL
LIN {X 0,Y 453.572,Z 383.989,A -85,B 0,C 180,E1 -8268.38,E2 -8268.38} C_VEL
LIN {X 0,Y 453.628,Z 383.979,A -85,B 0,C 180,E1 -8271.985,E2 -8271.985} C_VEL
LIN {X 0,Y 453.657,Z 383.977,A -85,B 0,C 180,E1 -8274.667,E2 -8274.667} C_VEL
LIN {X 0,Y 453.751,Z 383.965,A -85,B 0,C 180,E1 -8277.337,E2 -8277.337} C_VEL
LIN {X 0,Y 453.8,Z 383.958,A -85,B 0,C 180,E1 -8280,E2 -8280} C_VEL
LIN {X 0,Y 453.751,Z 383.964,A -85,B 0,C 180,E1 -8282.664,E2 -8282.664} C_VEL
LIN {X 0,Y 453.662,Z 383.973,A -85,B 0,C 180,E1 -8286.226,E2 -8286.226} C_VEL
LIN {X 0,Y 453.572,Z 383.986,A -85,B 0,C 180,E1 -8288.914,E2 -8288.914} C_VEL
LIN {X 0,Y 453.578,Z 383.985,A -85,B 0,C 180,E1 -8292.552,E2 -8292.552} C_VEL
LIN {X 0,Y 453.535,Z 383.99,A -85,B 0,C 180,E1 -8296.197,E2 -8296.197} C_VEL
LIN {X 0,Y 453.502,Z 383.993,A -85,B 0,C 180,E1 -8299.044,E2 -8299.044} C_VEL
LIN {X 0,Y 453.482,Z 383.996,A -85,B 0,C 180,E1 -8301.836,E2 -8301.836} C_VEL
LIN {X 0,Y 453.495,Z 383.996,A -85,B 0,C 180,E1 -8304.736,E2 -8304.736} C_VEL
LIN {X 0,Y 453.518,Z 383.993,A -85,B 0,C 180,E1 -8307.963,E2 -8307.963} C_VEL
LIN {X 0,Y 453.464,Z 383.999,A -85,B 0,C 180,E1 -8310.761,E2 -8310.761} C_VEL
LIN {X 0,Y 453.46,Z 384.003,A -85,B 0,C 180,E1 -8313.915,E2 -8313.915} C_VEL
LIN {X 0,Y 453.454,Z 384.002,A -85,B 0,C 180,E1 -8317.19,E2 -8317.19} C_VEL
LIN {X 0,Y 453.517,Z 383.996,A -85,B 0,C 180,E1 -8319.447,E2 -8319.447} C_VEL
LIN {X 0,Y 453.477,Z 384,A -85,B 0,C 180,E1 -8322.994,E2 -8322.994} C_VEL
LIN {X 0,Y 453.463,Z 384,A -85,B 0,C 180,E1 -8325.783,E2 -8325.783} C_VEL
LIN {X 0,Y 453.483,Z 383.999,A -85,B 0,C 180,E1 -8328.214,E2 -8328.214} C_VEL
LIN {X 0,Y 453.521,Z 383.994,A -85,B 0,C 180,E1 -8330.79,E2 -8330.79} C_VEL
LIN {X 0,Y 453.499,Z 384.062,A -85,B 0,C 180,E1 -8334.404,E2 -8334.404} C_VEL
LIN {X 0,Y 455.018,Z 391.686,A -85,B 0,C 180,E1 -8337.279,E2 -8337.279} C_VEL
LIN {X 0,Y 455.918,Z 397.764,A -85,B 0,C 180,E1 -8339.426,E2 -8339.426} C_VEL
LIN {X 0,Y 455.316,Z 405.791,A -85,B 0,C 180,E1 -8342.005,E2 -8342.005} C_VEL
LIN {X 0,Y 454.614,Z 416.569,A -85,B 0,C 180,E1 -8345.332,E2 -8345.332} C_VEL
LIN {X 0,Y 453.98,Z 427.845,A -85,B 0,C 180,E1 -8348.69,E2 -8348.69} C_VEL
LIN {X 0,Y 453.467,Z 439.117,A -85,B 0,C 180,E1 -8351.945,E2 -8351.945} C_VEL
LIN {X 0,Y 453.198,Z 447.579,A -85,B 0,C 180,E1 -8354.337,E2 -8354.337} C_VEL
LIN {X 0,Y 455.043,Z 461.66,A -85,B 0,C 180,E1 -8354.758,E2 -8354.758} C_VEL
LIN {X 0,Y 455.874,Z 469.77,A -85,B 0,C 180,E1 -8355.095,E2 -8355.095} C_VEL
LIN {X 0,Y 455.344,Z 482.166,A -85,B 0,C 180,E1 -8355.705,E2 -8355.705} C_VEL
LIN {X 0,Y 454.822,Z 494.017,A -85,B 0,C 180,E1 -8356.486,E2 -8356.486} C_VEL
LIN {X 0,Y 454.329,Z 504.124,A -85,B 0,C 180,E1 -8357.333,E2 -8357.333} C_VEL
LIN {X 0,Y 453.917,Z 514.318,A -85,B 0,C 180,E1 -8358.391,E2 -8358.391} C_VEL
LIN {X 0,Y 453.41,Z 523.125,A -85,B 0,C 180,E1 -8359.508,E2 -8359.508} C_VEL
LIN {X 0,Y 453.059,Z 531.665,A -85,B 0,C 180,E1 -8360.853,E2 -8360.853} C_VEL
LIN {X 0,Y 452.777,Z 538.524,A -85,B 0,C 180,E1 -8362.196,E2 -8362.196} C_VEL
LIN {X 0,Y 452.588,Z 544.298,A -85,B 0,C 180,E1 -8363.631,E2 -8363.631} C_VEL
LIN {X 0,Y 452.558,Z 548.825,A -85,B 0,C 180,E1 -8365.102,E2 -8365.102} C_VEL
LIN {X 0,Y 452.523,Z 551.865,A -85,B 0,C 180,E1 -8366.44,E2 -8366.44} C_VEL
LIN {X 0,Y 452.543,Z 553.331,A -85,B 0,C 180,E1 -8367.332,E2 -8367.332} C_VEL
LIN {X 0,Y 452.523,Z 554.357,A -85,B 0,C 180,E1 -8368.222,E2 -8368.222} C_VEL
LIN {X 0,Y 452.489,Z 554.967,A -85,B 0,C 180,E1 -8369.112,E2 -8369.112} C_VEL
LIN {X 0,Y 452.464,Z 555.176,A -85,B 0,C 180,E1 -8370.002,E2 -8370.002} C_VEL
LIN {X 0,Y 452.539,Z 554.324,A -85,B 0,C 180,E1 -8371.782,E2 -8371.782} C_VEL
LIN {X 0,Y 452.544,Z 553.325,A -85,B 0,C 180,E1 -8372.672,E2 -8372.672} C_VEL
LIN {X 0,Y 452.525,Z 551.871,A -85,B 0,C 180,E1 -8373.564,E2 -8373.564} C_VEL
LIN {X 0,Y 452.56,Z 548.888,A -85,B 0,C 180,E1 -8374.902,E2 -8374.902} C_VEL
LIN {X 0,Y 452.613,Z 544.299,A -85,B 0,C 180,E1 -8376.398,E2 -8376.398} C_VEL
LIN {X 0,Y 452.782,Z 538.607,A -85,B 0,C 180,E1 -8377.808,E2 -8377.808} C_VEL
LIN {X 0,Y 453.066,Z 531.775,A -85,B 0,C 180,E1 -8379.151,E2 -8379.151} C_VEL
LIN {X 0,Y 453.412,Z 523.233,A -85,B 0,C 180,E1 -8380.495,E2 -8380.495} C_VEL
LIN {X 0,Y 453.903,Z 514.428,A -85,B 0,C 180,E1 -8381.614,E2 -8381.614} C_VEL
LIN {X 0,Y 454.345,Z 504.183,A -85,B 0,C 180,E1 -8382.675,E2 -8382.675} C_VEL
LIN {X 0,Y 454.804,Z 494.106,A -85,B 0,C 180,E1 -8383.518,E2 -8383.518} C_VEL
LIN {X 0,Y 455.388,Z 482.22,A -85,B 0,C 180,E1 -8384.297,E2 -8384.297} C_VEL
LIN {X 0,Y 455.839,Z 469.774,A -85,B 0,C 180,E1 -8384.911,E2 -8384.911} C_VEL
LIN {X 0,Y 454.538,Z 457.083,A -85,B 0,C 180,E1 -8385.397,E2 -8385.397} C_VEL
LIN {X 0,Y 453.238,Z 447.764,A -85,B 0,C 180,E1 -8385.672,E2 -8385.672} C_VEL
LIN {X 0,Y 453.639,Z 435.746,A -85,B 0,C 180,E1 -8389.083,E2 -8389.083} C_VEL
LIN {X 0,Y 454.169,Z 424.688,A -85,B 0,C 180,E1 -8392.281,E2 -8392.281} C_VEL
LIN {X 0,Y 454.805,Z 413.405,A -85,B 0,C 180,E1 -8395.639,E2 -8395.639} C_VEL
LIN {X 0,Y 455.588,Z 402.195,A -85,B 0,C 180,E1 -8399.075,E2 -8399.075} C_VEL
LIN {X 0,Y 455.827,Z 397.425,A -85,B 0,C 180,E1 -8400.585,E2 -8400.585} C_VEL
LIN {X 0,Y 454.882,Z 391.079,A -85,B 0,C 180,E1 -8402.737,E2 -8402.737} C_VEL
LIN {X 0,Y 453.505,Z 383.997,A -85,B 0,C 180,E1 -8405.26,E2 -8405.26} C_VEL
LIN {X 0,Y 453.463,Z 384.003,A -85,B 0,C 180,E1 -8408.313,E2 -8408.313} C_VEL
LIN {X 0,Y 453.476,Z 383.997,A -85,B 0,C 180,E1 -8410.612,E2 -8410.612} C_VEL
LIN {X 0,Y 453.482,Z 383.996,A -85,B 0,C 180,E1 -8414.528,E2 -8414.528} C_VEL
LIN {X 0,Y 453.446,Z 384,A -85,B 0,C 180,E1 -8418.071,E2 -8418.071} C_VEL
LIN {X 0,Y 453.455,Z 384.002,A -85,B 0,C 180,E1 -8420.801,E2 -8420.801} C_VEL
LIN {X 0,Y 453.46,Z 384,A -85,B 0,C 180,E1 -8423.917,E2 -8423.917} C_VEL
LIN {X 0,Y 453.48,Z 383.996,A -85,B 0,C 180,E1 -8427.151,E2 -8427.151} C_VEL
LIN {X 0,Y 453.467,Z 383.998,A -85,B 0,C 180,E1 -8430.267,E2 -8430.267} C_VEL
LIN {X 0,Y 453.428,Z 384.006,A -85,B 0,C 180,E1 -8433.289,E2 -8433.289} C_VEL
LIN {X 0,Y 453.495,Z 383.994,A -85,B 0,C 180,E1 -8436.238,E2 -8436.238} C_VEL
LIN {X 0,Y 453.488,Z 383.997,A -85,B 0,C 180,E1 -8439.118,E2 -8439.118} C_VEL
LIN {X 0,Y 453.516,Z 383.995,A -85,B 0,C 180,E1 -8441.944,E2 -8441.944} C_VEL
LIN {X 0,Y 453.545,Z 383.99,A -85,B 0,C 180,E1 -8444.726,E2 -8444.726} C_VEL
LIN {X 0,Y 453.561,Z 383.988,A -85,B 0,C 180,E1 -8448.379,E2 -8448.379} C_VEL
LIN {X 0,Y 453.564,Z 383.989,A -85,B 0,C 180,E1 -8451.086,E2 -8451.086} C_VEL
LIN {X 0,Y 453.641,Z 383.978,A -85,B 0,C 180,E1 -8453.774,E2 -8453.774} C_VEL
LIN {X 0,Y 453.463,Z 384.001,A -85,B 0,C 180,E1 -8455.555,E2 -8455.555} C_VEL
LIN {X 0,Y 453.341,Z 384.127,A -85,B 0,C 180,E1 -8456.611,E2 -8456.611} C_VEL
LIN {X 0,Y 453.538,Z 389.937,A -85,B 0,C 180,E1 -8459.112,E2 -8459.112} C_VEL
LIN {X 0,Y 453.336,Z 396.08,A -85,B 0,C 180,E1 -8461.776,E2 -8461.776} C_VEL
LIN {X 0,Y 453.231,Z 404.089,A -85,B 0,C 180,E1 -8465.338,E2 -8465.338} C_VEL
LIN {X 0,Y 453.127,Z 410.029,A -85,B 0,C 180,E1 -8468.024,E2 -8468.024} C_VEL
LIN {X 0,Y 452.986,Z 416.017,A -85,B 0,C 180,E1 -8470.73,E2 -8470.73} C_VEL
LIN {X 0,Y 452.875,Z 421.957,A -85,B 0,C 180,E1 -8473.46,E2 -8473.46} C_VEL
LIN {X 0,Y 452.859,Z 425.617,A -85,B 0,C 180,E1 -8475.153,E2 -8475.153} C_VEL
LIN {X 0,Y 455.787,Z 439.905,A -85,B 0,C 180,E1 -8475.708,E2 -8475.708} C_VEL
LIN {X 0,Y 456.431,Z 445.273,A -85,B 0,C 180,E1 -8475.951,E2 -8475.951} C_VEL
LIN {X 0,Y 455.935,Z 457.707,A -85,B 0,C 180,E1 -8476.579,E2 -8476.579} C_VEL
LIN {X 0,Y 455.395,Z 469.931,A -85,B 0,C 180,E1 -8477.398,E2 -8477.398} C_VEL
LIN {X 0,Y 454.816,Z 481.071,A -85,B 0,C 180,E1 -8478.351,E2 -8478.351} C_VEL
LIN {X 0,Y 454.224,Z 492.04,A -85,B 0,C 180,E1 -8479.535,E2 -8479.535} C_VEL
LIN {X 0,Y 453.77,Z 500.288,A -85,B 0,C 180,E1 -8480.631,E2 -8480.631} C_VEL
LIN {X 0,Y 453.376,Z 507.77,A -85,B 0,C 180,E1 -8481.841,E2 -8481.841} C_VEL
LIN {X 0,Y 453.01,Z 514.85,A -85,B 0,C 180,E1 -8483.264,E2 -8483.264} C_VEL
LIN {X 0,Y 452.758,Z 520.766,A -85,B 0,C 180,E1 -8484.778,E2 -8484.778} C_VEL
LIN {X 0,Y 452.599,Z 525.123,A -85,B 0,C 180,E1 -8486.266,E2 -8486.266} C_VEL
LIN {X 0,Y 452.448,Z 528.223,A -85,B 0,C 180,E1 -8487.774,E2 -8487.774} C_VEL
LIN {X 0,Y 452.339,Z 530.345,A -85,B 0,C 180,E1 -8489.531,E2 -8489.531} C_VEL
LIN {X 0,Y 452.322,Z 530.867,A -85,B 0,C 180,E1 -8491.286,E2 -8491.286} C_VEL
LIN {X 0,Y 452.356,Z 529.923,A -85,B 0,C 180,E1 -8492.967,E2 -8492.967} C_VEL
LIN {X 0,Y 452.432,Z 527.66,A -85,B 0,C 180,E1 -8494.583,E2 -8494.583} C_VEL
LIN {X 0,Y 452.604,Z 524.052,A -85,B 0,C 180,E1 -8496.161,E2 -8496.161} C_VEL
LIN {X 0,Y 452.812,Z 519.263,A -85,B 0,C 180,E1 -8497.667,E2 -8497.667} C_VEL
LIN {X 0,Y 453.068,Z 513.137,A -85,B 0,C 180,E1 -8499.139,E2 -8499.139} C_VEL
LIN {X 0,Y 453.409,Z 505.23,A -85,B 0,C 180,E1 -8500.618,E2 -8500.618} C_VEL
LIN {X 0,Y 453.817,Z 497.737,A -85,B 0,C 180,E1 -8501.752,E2 -8501.752} C_VEL
LIN {X 0,Y 454.332,Z 488.602,A -85,B 0,C 180,E1 -8502.892,E2 -8502.892} C_VEL
LIN {X 0,Y 454.867,Z 478.176,A -85,B 0,C 180,E1 -8503.942,E2 -8503.942} C_VEL
LIN {X 0,Y 455.412,Z 466.933,A -85,B 0,C 180,E1 -8504.852,E2 -8504.852} C_VEL
LIN {X 0,Y 455.873,Z 455.849,A -85,B 0,C 180,E1 -8505.559,E2 -8505.559} C_VEL
LIN {X 0,Y 456.306,Z 444.23,A -85,B 0,C 180,E1 -8506.124,E2 -8506.124} C_VEL
LIN {X 0,Y 454.464,Z 433.41,A -85,B 0,C 180,E1 -8506.582,E2 -8506.582} C_VEL
LIN {X 0,Y 452.808,Z 425.186,A -85,B 0,C 180,E1 -8506.869,E2 -8506.869} C_VEL
LIN {X 0,Y 452.909,Z 418.515,A -85,B 0,C 180,E1 -8509.999,E2 -8509.999} C_VEL
LIN {X 0,Y 453.004,Z 411.468,A -85,B 0,C 180,E1 -8513.308,E2 -8513.308} C_VEL
LIN {X 0,Y 453.163,Z 405.602,A -85,B 0,C 180,E1 -8516.059,E2 -8516.059} C_VEL
LIN {X 0,Y 453.298,Z 398.851,A -85,B 0,C 180,E1 -8519.226,E2 -8519.226} C_VEL
LIN {X 0,Y 453.335,Z 392.313,A -85,B 0,C 180,E1 -8522.283,E2 -8522.283} C_VEL
LIN {X 0,Y 453.509,Z 385.958,A -85,B 0,C 180,E1 -8525.264,E2 -8525.264} C_VEL
LIN {X 0,Y 453.588,Z 383.987,A -85,B 0,C 180,E1 -8526.242,E2 -8526.242} C_VEL
LIN {X 0,Y 453.505,Z 383.995,A -85,B 0,C 180,E1 -8530.065,E2 -8530.065} C_VEL
LIN {X 0,Y 453.497,Z 383.994,A -85,B 0,C 180,E1 -8530.456,E2 -8530.456} C_VEL
LIN {X 0,Y 452.839,Z 384.078,A -85,B 0,C 180,E1 -8531.197,E2 -8531.197} C_VEL
LIN {X 0,Y 449.985,Z 384.434,A -85,B 0,C 180,E1 -8532.401,E2 -8532.401} C_VEL
LIN {X 0,Y 447.582,Z 384.734,A -85,B 0,C 180,E1 -8533.372,E2 -8533.372} C_VEL
LIN {X 0,Y 446.573,Z 384.858,A -85,B 0,C 180,E1 -8534.122,E2 -8534.122} C_VEL
LIN {X 0,Y 446.504,Z 384.865,A -85,B 0,C 180,E1 -8534.376,E2 -8534.376} C_VEL
LIN {X 0,Y 446.517,Z 384.865,A -85,B 0,C 180,E1 -8537.382,E2 -8537.382} C_VEL
LIN {X 0,Y 446.537,Z 384.863,A -85,B 0,C 180,E1 -8540.943,E2 -8540.943} C_VEL
LIN {X 0,Y 446.619,Z 384.854,A -85,B 0,C 180,E1 -8543.674,E2 -8543.674} C_VEL
LIN {X 0,Y 446.654,Z 384.849,A -85,B 0,C 180,E1 -8547.292,E2 -8547.292} C_VEL
LIN {X 0,Y 446.788,Z 384.964,A -85,B 0,C 180,E1 -8549.547,E2 -8549.547} C_VEL
LIN {X 0,Y 446.637,Z 388.844,A -85,B 0,C 180,E1 -8551.801,E2 -8551.801} C_VEL
LIN {X 0,Y 446.483,Z 395.18,A -85,B 0,C 180,E1 -8555.417,E2 -8555.417} C_VEL
LIN {X 0,Y 446.251,Z 400.056,A -85,B 0,C 180,E1 -8558.146,E2 -8558.146} C_VEL
LIN {X 0,Y 446.074,Z 406.709,A -85,B 0,C 180,E1 -8561.817,E2 -8561.817} C_VEL
LIN {X 0,Y 445.815,Z 413.557,A -85,B 0,C 180,E1 -8565.542,E2 -8565.542} C_VEL
LIN {X 0,Y 445.662,Z 419.805,A -85,B 0,C 180,E1 -8568.883,E2 -8568.883} C_VEL
LIN {X 0,Y 445.651,Z 422.074,A -85,B 0,C 180,E1 -8570.087,E2 -8570.087} C_VEL
LIN {X 0,Y 447.886,Z 434.317,A -85,B 0,C 180,E1 -8570.612,E2 -8570.612} C_VEL
LIN {X 0,Y 448.39,Z 439.646,A -85,B 0,C 180,E1 -8570.888,E2 -8570.888} C_VEL
LIN {X 0,Y 447.946,Z 450.028,A -85,B 0,C 180,E1 -8571.512,E2 -8571.512} C_VEL
LIN {X 0,Y 447.44,Z 460.953,A -85,B 0,C 180,E1 -8572.387,E2 -8572.387} C_VEL
LIN {X 0,Y 447.001,Z 470.535,A -85,B 0,C 180,E1 -8573.388,E2 -8573.388} C_VEL
LIN {X 0,Y 446.645,Z 478.066,A -85,B 0,C 180,E1 -8574.369,E2 -8574.369} C_VEL
LIN {X 0,Y 446.25,Z 485.763,A -85,B 0,C 180,E1 -8575.635,E2 -8575.635} C_VEL
LIN {X 0,Y 445.902,Z 491.938,A -85,B 0,C 180,E1 -8576.942,E2 -8576.942} C_VEL
LIN {X 0,Y 445.715,Z 496.564,A -85,B 0,C 180,E1 -8578.229,E2 -8578.229} C_VEL
LIN {X 0,Y 445.652,Z 499.385,A -85,B 0,C 180,E1 -8579.264,E2 -8579.264} C_VEL
LIN {X 0,Y 445.507,Z 501.524,A -85,B 0,C 180,E1 -8580.316,E2 -8580.316} C_VEL
LIN {X 0,Y 445.369,Z 503.141,A -85,B 0,C 180,E1 -8581.557,E2 -8581.557} C_VEL
LIN {X 0,Y 445.332,Z 503.744,A -85,B 0,C 180,E1 -8582.447,E2 -8582.447} C_VEL
LIN {X 0,Y 445.347,Z 503.801,A -85,B 0,C 180,E1 -8583.524,E2 -8583.524} C_VEL
LIN {X 0,Y 445.456,Z 502.909,A -85,B 0,C 180,E1 -8584.875,E2 -8584.875} C_VEL
LIN {X 0,Y 445.59,Z 500.443,A -85,B 0,C 180,E1 -8586.449,E2 -8586.449} C_VEL
LIN {X 0,Y 445.827,Z 496.463,A -85,B 0,C 180,E1 -8587.983,E2 -8587.983} C_VEL
LIN {X 0,Y 445.995,Z 492.611,A -85,B 0,C 180,E1 -8589.07,E2 -8589.07} C_VEL
LIN {X 0,Y 446.237,Z 487.479,A -85,B 0,C 180,E1 -8590.216,E2 -8590.216} C_VEL
LIN {X 0,Y 446.591,Z 480.979,A -85,B 0,C 180,E1 -8591.369,E2 -8591.369} C_VEL
LIN {X 0,Y 446.973,Z 472.671,A -85,B 0,C 180,E1 -8592.537,E2 -8592.537} C_VEL
LIN {X 0,Y 447.479,Z 463.42,A -85,B 0,C 180,E1 -8593.554,E2 -8593.554} C_VEL
LIN {X 0,Y 447.957,Z 453.859,A -85,B 0,C 180,E1 -8594.385,E2 -8594.385} C_VEL
LIN {X 0,Y 448.446,Z 442.185,A -85,B 0,C 180,E1 -8595.152,E2 -8595.152} C_VEL
LIN {X 0,Y 448.349,Z 436.436,A -85,B 0,C 180,E1 -8595.455,E2 -8595.455} C_VEL
LIN {X 0,Y 446.107,Z 424.559,A -85,B 0,C 180,E1 -8596.001,E2 -8596.001} C_VEL
LIN {X 0,Y 445.716,Z 422.452,A -85,B 0,C 180,E1 -8596.101,E2 -8596.101} C_VEL
LIN {X 0,Y 445.776,Z 416.774,A -85,B 0,C 180,E1 -8599.174,E2 -8599.174} C_VEL
LIN {X 0,Y 445.919,Z 411.46,A -85,B 0,C 180,E1 -8602.073,E2 -8602.073} C_VEL
LIN {X 0,Y 446.061,Z 406.164,A -85,B 0,C 180,E1 -8605.009,E2 -8605.009} C_VEL
LIN {X 0,Y 446.269,Z 400.382,A -85,B 0,C 180,E1 -8608.25,E2 -8608.25} C_VEL
LIN {X 0,Y 446.402,Z 395.929,A -85,B 0,C 180,E1 -8610.788,E2 -8610.788} C_VEL
LIN {X 0,Y 446.661,Z 390.561,A -85,B 0,C 180,E1 -8613.86,E2 -8613.86} C_VEL
LIN {X 0,Y 446.719,Z 387.175,A -85,B 0,C 180,E1 -8615.855,E2 -8615.855} C_VEL
LIN {X 0,Y 446.499,Z 384.872,A -85,B 0,C 180,E1 -8617.317,E2 -8617.317} C_VEL
LIN {X 0,Y 446.451,Z 384.879,A -85,B 0,C 180,E1 -8620.814,E2 -8620.814} C_VEL
LIN {X 0,Y 446.471,Z 384.875,A -85,B 0,C 180,E1 -8623.771,E2 -8623.771} C_VEL
LIN {X 0,Y 446.529,Z 384.866,A -85,B 0,C 180,E1 -8627.362,E2 -8627.362} C_VEL
LIN {X 0,Y 446.52,Z 384.867,A -85,B 0,C 180,E1 -8630.945,E2 -8630.945} C_VEL
LIN {X 0,Y 446.629,Z 384.854,A -85,B 0,C 180,E1 -8633.676,E2 -8633.676} C_VEL
LIN {X 0,Y 446.695,Z 384.844,A -85,B 0,C 180,E1 -8637.295,E2 -8637.295} C_VEL
LIN {X 0,Y 446.77,Z 384.834,A -85,B 0,C 180,E1 -8640,E2 -8640} C_VEL
LIN {X 0,Y 446.695,Z 384.843,A -85,B 0,C 180,E1 -8642.706,E2 -8642.706} C_VEL
LIN {X 0,Y 446.629,Z 384.849,A -85,B 0,C 180,E1 -8646.324,E2 -8646.324} C_VEL
LIN {X 0,Y 446.518,Z 384.863,A -85,B 0,C 180,E1 -8649.056,E2 -8649.056} C_VEL
LIN {X 0,Y 446.512,Z 384.865,A -85,B 0,C 180,E1 -8652.73,E2 -8652.73} C_VEL
LIN {X 0,Y 446.475,Z 384.87,A -85,B 0,C 180,E1 -8656.46,E2 -8656.46} C_VEL
LIN {X 0,Y 446.45,Z 384.874,A -85,B 0,C 180,E1 -8659.304,E2 -8659.304} C_VEL
LIN {X 0,Y 446.42,Z 384.879,A -85,B 0,C 180,E1 -8662.2,E2 -8662.2} C_VEL
LIN {X 0,Y 446.438,Z 384.875,A -85,B 0,C 180,E1 -8665.154,E2 -8665.154} C_VEL
LIN {X 0,Y 446.464,Z 384.871,A -85,B 0,C 180,E1 -8668.18,E2 -8668.18} C_VEL
LIN {X 0,Y 446.401,Z 384.882,A -85,B 0,C 180,E1 -8671.302,E2 -8671.302} C_VEL
LIN {X 0,Y 446.412,Z 384.879,A -85,B 0,C 180,E1 -8674.525,E2 -8674.525} C_VEL
LIN {X 0,Y 446.422,Z 384.88,A -85,B 0,C 180,E1 -8678.085,E2 -8678.085} C_VEL
LIN {X 0,Y 446.432,Z 384.878,A -85,B 0,C 180,E1 -8680.923,E2 -8680.923} C_VEL
LIN {X 0,Y 446.431,Z 384.877,A -85,B 0,C 180,E1 -8683.843,E2 -8683.843} C_VEL
LIN {X 0,Y 446.433,Z 384.877,A -85,B 0,C 180,E1 -8686.399,E2 -8686.399} C_VEL
LIN {X 0,Y 446.457,Z 384.874,A -85,B 0,C 180,E1 -8689.807,E2 -8689.807} C_VEL
LIN {X 0,Y 446.423,Z 384.878,A -85,B 0,C 180,E1 -8692.126,E2 -8692.126} C_VEL
LIN {X 0,Y 446.41,Z 384.912,A -85,B 0,C 180,E1 -8694.029,E2 -8694.029} C_VEL
LIN {X 0,Y 447.808,Z 391.729,A -85,B 0,C 180,E1 -8696.685,E2 -8696.685} C_VEL
LIN {X 0,Y 448.875,Z 397.788,A -85,B 0,C 180,E1 -8698.893,E2 -8698.893} C_VEL
LIN {X 0,Y 448.765,Z 402.373,A -85,B 0,C 180,E1 -8700.444,E2 -8700.444} C_VEL
LIN {X 0,Y 447.867,Z 413.321,A -85,B 0,C 180,E1 -8703.939,E2 -8703.939} C_VEL
LIN {X 0,Y 447.223,Z 422.78,A -85,B 0,C 180,E1 -8706.87,E2 -8706.87} C_VEL
LIN {X 0,Y 446.739,Z 432.425,A -85,B 0,C 180,E1 -8709.754,E2 -8709.754} C_VEL
LIN {X 0,Y 446.247,Z 443.739,A -85,B 0,C 180,E1 -8713.063,E2 -8713.063} C_VEL
LIN {X 0,Y 446.153,Z 447.332,A -85,B 0,C 180,E1 -8714.093,E2 -8714.093} C_VEL
LIN {X 0,Y 448.103,Z 461.552,A -85,B 0,C 180,E1 -8714.539,E2 -8714.539} C_VEL
LIN {X 0,Y 448.932,Z 470.421,A -85,B 0,C 180,E1 -8714.917,E2 -8714.917} C_VEL
LIN {X 0,Y 448.453,Z 481.593,A -85,B 0,C 180,E1 -8715.481,E2 -8715.481} C_VEL
LIN {X 0,Y 447.886,Z 493.515,A -85,B 0,C 180,E1 -8716.273,E2 -8716.273} C_VEL
LIN {X 0,Y 447.328,Z 504.15,A -85,B 0,C 180,E1 -8717.18,E2 -8717.18} C_VEL
LIN {X 0,Y 446.917,Z 513.866,A -85,B 0,C 180,E1 -8718.206,E2 -8718.206} C_VEL
LIN {X 0,Y 446.372,Z 522.691,A -85,B 0,C 180,E1 -8719.341,E2 -8719.341} C_VEL
LIN {X 0,Y 446.02,Z 531.239,A -85,B 0,C 180,E1 -8720.708,E2 -8720.708} C_VEL
LIN {X 0,Y 445.715,Z 538.197,A -85,B 0,C 180,E1 -8722.072,E2 -8722.072} C_VEL
LIN {X 0,Y 445.489,Z 544.5,A -85,B 0,C 180,E1 -8723.662,E2 -8723.662} C_VEL
LIN {X 0,Y 445.489,Z 548.617,A -85,B 0,C 180,E1 -8725.024,E2 -8725.024} C_VEL
LIN {X 0,Y 445.419,Z 551.663,A -85,B 0,C 180,E1 -8726.384,E2 -8726.384} C_VEL
LIN {X 0,Y 445.466,Z 553.127,A -85,B 0,C 180,E1 -8727.289,E2 -8727.289} C_VEL
LIN {X 0,Y 445.437,Z 554.155,A -85,B 0,C 180,E1 -8728.194,E2 -8728.194} C_VEL
LIN {X 0,Y 445.397,Z 554.774,A -85,B 0,C 180,E1 -8729.098,E2 -8729.098} C_VEL
LIN {X 0,Y 445.371,Z 554.984,A -85,B 0,C 180,E1 -8730.002,E2 -8730.002} C_VEL
LIN {X 0,Y 445.398,Z 554.758,A -85,B 0,C 180,E1 -8730.906,E2 -8730.906} C_VEL
LIN {X 0,Y 445.451,Z 554.137,A -85,B 0,C 180,E1 -8731.81,E2 -8731.81} C_VEL
LIN {X 0,Y 445.467,Z 553.109,A -85,B 0,C 180,E1 -8732.715,E2 -8732.715} C_VEL
LIN {X 0,Y 445.422,Z 551.63,A -85,B 0,C 180,E1 -8733.62,E2 -8733.62} C_VEL
LIN {X 0,Y 445.491,Z 548.588,A -85,B 0,C 180,E1 -8734.98,E2 -8734.98} C_VEL
LIN {X 0,Y 445.532,Z 544.313,A -85,B 0,C 180,E1 -8736.387,E2 -8736.387} C_VEL
LIN {X 0,Y 445.719,Z 538.175,A -85,B 0,C 180,E1 -8737.932,E2 -8737.932} C_VEL
LIN {X 0,Y 446.026,Z 531.317,A -85,B 0,C 180,E1 -8739.296,E2 -8739.296} C_VEL
LIN {X 0,Y 446.374,Z 522.757,A -85,B 0,C 180,E1 -8740.663,E2 -8740.663} C_VEL
LIN {X 0,Y 446.908,Z 513.928,A -85,B 0,C 180,E1 -8741.798,E2 -8741.798} C_VEL
LIN {X 0,Y 447.347,Z 504.16,A -85,B 0,C 180,E1 -8742.827,E2 -8742.827} C_VEL
LIN {X 0,Y 447.867,Z 493.463,A -85,B 0,C 180,E1 -8743.732,E2 -8743.732} C_VEL
LIN {X 0,Y 448.478,Z 481.505,A -85,B 0,C 180,E1 -8744.523,E2 -8744.523} C_VEL
LIN {X 0,Y 448.905,Z 468.94,A -85,B 0,C 180,E1 -8745.146,E2 -8745.146} C_VEL
LIN {X 0,Y 447.154,Z 454.277,A -85,B 0,C 180,E1 -8745.719,E2 -8745.719} C_VEL
LIN {X 0,Y 446.179,Z 447.437,A -85,B 0,C 180,E1 -8745.93,E2 -8745.93} C_VEL
LIN {X 0,Y 446.598,Z 435.79,A -85,B 0,C 180,E1 -8749.299,E2 -8749.299} C_VEL
LIN {X 0,Y 447.174,Z 424.479,A -85,B 0,C 180,E1 -8752.649,E2 -8752.649} C_VEL
LIN {X 0,Y 447.772,Z 414.842,A -85,B 0,C 180,E1 -8755.572,E2 -8755.572} C_VEL
LIN {X 0,Y 448.613,Z 403.658,A -85,B 0,C 180,E1 -8759.056,E2 -8759.056} C_VEL
LIN {X 0,Y 448.87,Z 399.012,A -85,B 0,C 180,E1 -8760.555,E2 -8760.555} C_VEL
LIN {X 0,Y 448.251,Z 394.144,A -85,B 0,C 180,E1 -8762.215,E2 -8762.215} C_VEL
LIN {X 0,Y 446.494,Z 385.122,A -85,B 0,C 180,E1 -8765.467,E2 -8765.467} C_VEL
LIN {X 0,Y 446.442,Z 384.876,A -85,B 0,C 180,E1 -8765.625,E2 -8765.625} C_VEL
LIN {X 0,Y 446.414,Z 384.878,A -85,B 0,C 180,E1 -8769.032,E2 -8769.032} C_VEL
LIN {X 0,Y 446.385,Z 384.882,A -85,B 0,C 180,E1 -8772.27,E2 -8772.27} C_VEL
LIN {X 0,Y 446.426,Z 384.878,A -85,B 0,C 180,E1 -8775.108,E2 -8775.108} C_VEL
LIN {X 0,Y 446.408,Z 384.879,A -85,B 0,C 180,E1 -8778.606,E2 -8778.606} C_VEL
LIN {X 0,Y 446.418,Z 384.873,A -85,B 0,C 180,E1 -8781.922,E2 -8781.922} C_VEL
LIN {X 0,Y 446.429,Z 384.875,A -85,B 0,C 180,E1 -8785.477,E2 -8785.477} C_VEL
LIN {X 0,Y 446.417,Z 384.875,A -85,B 0,C 180,E1 -8788.699,E2 -8788.699} C_VEL
LIN {X 0,Y 446.429,Z 384.877,A -85,B 0,C 180,E1 -8791.836,E2 -8791.836} C_VEL
LIN {X 0,Y 446.417,Z 384.879,A -85,B 0,C 180,E1 -8794.845,E2 -8794.845} C_VEL
LIN {X 0,Y 446.454,Z 384.873,A -85,B 0,C 180,E1 -8798.245,E2 -8798.245} C_VEL
LIN {X 0,Y 446.462,Z 384.871,A -85,B 0,C 180,E1 -8801.649,E2 -8801.649} C_VEL
LIN {X 0,Y 446.513,Z 384.868,A -85,B 0,C 180,E1 -8804.48,E2 -8804.48} C_VEL
LIN {X 0,Y 446.52,Z 384.866,A -85,B 0,C 180,E1 -8808.193,E2 -8808.193} C_VEL
LIN {X 0,Y 446.515,Z 384.867,A -85,B 0,C 180,E1 -8810.944,E2 -8810.944} C_VEL
LIN {X 0,Y 446.611,Z 384.855,A -85,B 0,C 180,E1 -8813.675,E2 -8813.675} C_VEL
LIN {X 0,Y 446.429,Z 384.878,A -85,B 0,C 180,E1 -8815.485,E2 -8815.485} C_VEL
LIN {X 0,Y 446.299,Z 385.043,A -85,B 0,C 180,E1 -8816.501,E2 -8816.501} C_VEL
LIN {X 0,Y 446.54,Z 391.016,A -85,B 0,C 180,E1 -8819.098,E2 -8819.098} C_VEL
LIN {X 0,Y 446.297,Z 397.19,A -85,B 0,C 180,E1 -8821.805,E2 -8821.805} C_VEL
LIN {X 0,Y 446.187,Z 405.207,A -85,B 0,C 180,E1 -8825.423,E2 -8825.423} C_VEL
LIN {X 0,Y 446.072,Z 411.245,A -85,B 0,C 180,E1 -8828.152,E2 -8828.152} C_VEL
LIN {X 0,Y 445.938,Z 417.239,A -85,B 0,C 180,E1 -8830.901,E2 -8830.901} C_VEL
LIN {X 0,Y 445.798,Z 423.228,A -85,B 0,C 180,E1 -8833.678,E2 -8833.678} C_VEL
LIN {X 0,Y 445.798,Z 425.791,A -85,B 0,C 180,E1 -8834.872,E2 -8834.872} C_VEL
LIN {X 0,Y 448.96,Z 441.045,A -85,B 0,C 180,E1 -8835.491,E2 -8835.491} C_VEL
LIN {X 0,Y 449.56,Z 446.725,A -85,B 0,C 180,E1 -8835.761,E2 -8835.761} C_VEL
LIN {X 0,Y 448.986,Z 459.797,A -85,B 0,C 180,E1 -8836.46,E2 -8836.46} C_VEL
LIN {X 0,Y 448.489,Z 470.503,A -85,B 0,C 180,E1 -8837.207,E2 -8837.207} C_VEL
LIN {X 0,Y 447.874,Z 481.526,A -85,B 0,C 180,E1 -8838.172,E2 -8838.172} C_VEL
LIN {X 0,Y 447.325,Z 491.538,A -85,B 0,C 180,E1 -8839.264,E2 -8839.264} C_VEL
LIN {X 0,Y 446.788,Z 500.662,A -85,B 0,C 180,E1 -8840.487,E2 -8840.487} C_VEL
LIN {X 0,Y 446.281,Z 509.191,A -85,B 0,C 180,E1 -8841.919,E2 -8841.919} C_VEL
LIN {X 0,Y 445.954,Z 515.349,A -85,B 0,C 180,E1 -8843.202,E2 -8843.202} C_VEL
LIN {X 0,Y 445.68,Z 521.07,A -85,B 0,C 180,E1 -8844.701,E2 -8844.701} C_VEL
LIN {X 0,Y 445.537,Z 525.385,A -85,B 0,C 180,E1 -8846.211,E2 -8846.211} C_VEL
LIN {X 0,Y 445.335,Z 528.712,A -85,B 0,C 180,E1 -8847.899,E2 -8847.899} C_VEL
LIN {X 0,Y 445.25,Z 530.706,A -85,B 0,C 180,E1 -8849.755,E2 -8849.755} C_VEL
LIN {X 0,Y 445.234,Z 531.012,A -85,B 0,C 180,E1 -8851.526,E2 -8851.526} C_VEL
LIN {X 0,Y 445.268,Z 529.883,A -85,B 0,C 180,E1 -8853.222,E2 -8853.222} C_VEL
LIN {X 0,Y 445.39,Z 527.388,A -85,B 0,C 180,E1 -8854.861,E2 -8854.861} C_VEL
LIN {X 0,Y 445.56,Z 523.659,A -85,B 0,C 180,E1 -8856.442,E2 -8856.442} C_VEL
LIN {X 0,Y 445.768,Z 518.68,A -85,B 0,C 180,E1 -8857.971,E2 -8857.971} C_VEL
LIN {X 0,Y 446.062,Z 512.299,A -85,B 0,C 180,E1 -8859.462,E2 -8859.462} C_VEL
LIN {X 0,Y 446.472,Z 504.404,A -85,B 0,C 180,E1 -8860.923,E2 -8860.923} C_VEL
LIN {X 0,Y 446.897,Z 496.095,A -85,B 0,C 180,E1 -8862.154,E2 -8862.154} C_VEL
LIN {X 0,Y 447.493,Z 485.673,A -85,B 0,C 180,E1 -8863.401,E2 -8863.401} C_VEL
LIN {X 0,Y 448.06,Z 474.988,A -85,B 0,C 180,E1 -8864.428,E2 -8864.428} C_VEL
LIN {X 0,Y 448.589,Z 463.873,A -85,B 0,C 180,E1 -8865.276,E2 -8865.276} C_VEL
LIN {X 0,Y 449.215,Z 451.171,A -85,B 0,C 180,E1 -8866.027,E2 -8866.027} C_VEL
LIN {X 0,Y 449.287,Z 443.805,A -85,B 0,C 180,E1 -8866.371,E2 -8866.371} C_VEL
LIN {X 0,Y 446.889,Z 430.978,A -85,B 0,C 180,E1 -8866.911,E2 -8866.911} C_VEL
LIN {X 0,Y 445.742,Z 425.31,A -85,B 0,C 180,E1 -8867.12,E2 -8867.12} C_VEL
LIN {X 0,Y 445.864,Z 418.022,A -85,B 0,C 180,E1 -8870.567,E2 -8870.567} C_VEL
LIN {X 0,Y 445.963,Z 411.843,A -85,B 0,C 180,E1 -8873.486,E2 -8873.486} C_VEL
LIN {X 0,Y 446.113,Z 405.246,A -85,B 0,C 180,E1 -8876.611,E2 -8876.611} C_VEL
LIN {X 0,Y 446.232,Z 398.631,A -85,B 0,C 180,E1 -8879.734,E2 -8879.734} C_VEL
LIN {X 0,Y 446.3,Z 392.09,A -85,B 0,C 180,E1 -8882.826,E2 -8882.826} C_VEL
LIN {X 0,Y 446.555,Z 384.863,A -85,B 0,C 180,E1 -8886.253,E2 -8886.253} C_VEL
LIN {X 0,Y 446.446,Z 384.873,A -85,B 0,C 180,E1 -8889.736,E2 -8889.736} C_VEL
LIN {X 0,Y 446.457,Z 384.872,A -85,B 0,C 180,E1 -8892.595,E2 -8892.595} C_VEL
LIN {X 0,Y 446.504,Z 384.865,A -85,B 0,C 180,E1 -8894.376,E2 -8894.376} C_VEL
LIN {X 0,Y 445.875,Z 384.948,A -85,B 0,C 180,E1 -8895.129,E2 -8895.129} C_VEL
LIN {X 0,Y 443.045,Z 385.299,A -85,B 0,C 180,E1 -8896.353,E2 -8896.353} C_VEL
LIN {X 0,Y 440.615,Z 385.602,A -85,B 0,C 180,E1 -8897.339,E2 -8897.339} C_VEL
LIN {X 0,Y 439.549,Z 385.735,A -85,B 0,C 180,E1 -8898.102,E2 -8898.102} C_VEL
LIN {X 0,Y 439.451,Z 385.744,A -85,B 0,C 180,E1 -8898.36,E2 -8898.36} C_VEL
LIN {X 0,Y 439.533,Z 385.737,A -85,B 0,C 180,E1 -8901.724,E2 -8901.724} C_VEL
LIN {X 0,Y 439.608,Z 385.73,A -85,B 0,C 180,E1 -8904.494,E2 -8904.494} C_VEL
LIN {X 0,Y 439.627,Z 385.726,A -85,B 0,C 180,E1 -8908.166,E2 -8908.166} C_VEL
LIN {X 0,Y 439.735,Z 385.805,A -85,B 0,C 180,E1 -8909.426,E2 -8909.426} C_VEL
LIN {X 0,Y 439.768,Z 388.329,A -85,B 0,C 180,E1 -8910.914,E2 -8910.914} C_VEL
LIN {X 0,Y 439.376,Z 394.656,A -85,B 0,C 180,E1 -8914.585,E2 -8914.585} C_VEL
LIN {X 0,Y 439.296,Z 399.513,A -85,B 0,C 180,E1 -8917.351,E2 -8917.351} C_VEL
LIN {X 0,Y 439.022,Z 406.161,A -85,B 0,C 180,E1 -8921.073,E2 -8921.073} C_VEL
LIN {X 0,Y 438.902,Z 409.555,A -85,B 0,C 180,E1 -8922.952,E2 -8922.952} C_VEL
LIN {X 0,Y 438.737,Z 415.185,A -85,B 0,C 180,E1 -8926.03,E2 -8926.03} C_VEL
LIN {X 0,Y 438.605,Z 422.375,A -85,B 0,C 180,E1 -8929.874,E2 -8929.874} C_VEL
LIN {X 0,Y 440.701,Z 433.737,A -85,B 0,C 180,E1 -8930.353,E2 -8930.353} C_VEL
LIN {X 0,Y 441.482,Z 439.886,A -85,B 0,C 180,E1 -8930.681,E2 -8930.681} C_VEL
LIN {X 0,Y 441.082,Z 449.351,A -85,B 0,C 180,E1 -8931.25,E2 -8931.25} C_VEL
LIN {X 0,Y 440.521,Z 459.591,A -85,B 0,C 180,E1 -8932.056,E2 -8932.056} C_VEL
LIN {X 0,Y 440.093,Z 469.205,A -85,B 0,C 180,E1 -8933.029,E2 -8933.029} C_VEL
LIN {X 0,Y 439.645,Z 478.464,A -85,B 0,C 180,E1 -8934.231,E2 -8934.231} C_VEL
LIN {X 0,Y 439.196,Z 486.569,A -85,B 0,C 180,E1 -8935.595,E2 -8935.595} C_VEL
LIN {X 0,Y 438.856,Z 492.52,A -85,B 0,C 180,E1 -8936.895,E2 -8936.895} C_VEL
LIN {X 0,Y 438.639,Z 497.136,A -85,B 0,C 180,E1 -8938.21,E2 -8938.21} C_VEL
LIN {X 0,Y 438.512,Z 501.034,A -85,B 0,C 180,E1 -8939.788,E2 -8939.788} C_VEL
LIN {X 0,Y 438.337,Z 502.801,A -85,B 0,C 180,E1 -8940.865,E2 -8940.865} C_VEL
LIN {X 0,Y 438.265,Z 503.88,A -85,B 0,C 180,E1 -8941.947,E2 -8941.947} C_VEL
LIN {X 0,Y 438.267,Z 504.212,A -85,B 0,C 180,E1 -8943.503,E2 -8943.503} C_VEL
LIN {X 0,Y 438.392,Z 503.024,A -85,B 0,C 180,E1 -8945.156,E2 -8945.156} C_VEL
LIN {X 0,Y 438.536,Z 500.361,A -85,B 0,C 180,E1 -8946.746,E2 -8946.746} C_VEL
LIN {X 0,Y 438.8,Z 496.177,A -85,B 0,C 180,E1 -8948.298,E2 -8948.298} C_VEL
LIN {X 0,Y 439.028,Z 491.665,A -85,B 0,C 180,E1 -8949.514,E2 -8949.514} C_VEL
LIN {X 0,Y 439.327,Z 486.153,A -85,B 0,C 180,E1 -8950.68,E2 -8950.68} C_VEL
LIN {X 0,Y 439.718,Z 478.834,A -85,B 0,C 180,E1 -8951.913,E2 -8951.913} C_VEL
LIN {X 0,Y 440.13,Z 471.039,A -85,B 0,C 180,E1 -8952.952,E2 -8952.952} C_VEL
LIN {X 0,Y 440.645,Z 462.031,A -85,B 0,C 180,E1 -8953.916,E2 -8953.916} C_VEL
LIN {X 0,Y 441.204,Z 451.179,A -85,B 0,C 180,E1 -8954.814,E2 -8954.814} C_VEL
LIN {X 0,Y 441.61,Z 440.443,A -85,B 0,C 180,E1 -8955.485,E2 -8955.485} C_VEL
LIN {X 0,Y 441.194,Z 435.883,A -85,B 0,C 180,E1 -8955.732,E2 -8955.732} C_VEL
LIN {X 0,Y 438.93,Z 424.289,A -85,B 0,C 180,E1 -8956.268,E2 -8956.268} C_VEL
LIN {X 0,Y 438.642,Z 422.712,A -85,B 0,C 180,E1 -8956.327,E2 -8956.327} C_VEL
LIN {X 0,Y 438.735,Z 416.857,A -85,B 0,C 180,E1 -8959.552,E2 -8959.552} C_VEL
LIN {X 0,Y 438.909,Z 411.492,A -85,B 0,C 180,E1 -8962.521,E2 -8962.521} C_VEL
LIN {X 0,Y 439.013,Z 407.421,A -85,B 0,C 180,E1 -8964.809,E2 -8964.809} C_VEL
LIN {X 0,Y 439.219,Z 401.558,A -85,B 0,C 180,E1 -8968.127,E2 -8968.127} C_VEL
LIN {X 0,Y 439.43,Z 396.006,A -85,B 0,C 180,E1 -8971.328,E2 -8971.328} C_VEL
LIN {X 0,Y 439.654,Z 390.723,A -85,B 0,C 180,E1 -8974.431,E2 -8974.431} C_VEL
LIN {X 0,Y 439.653,Z 387.346,A -85,B 0,C 180,E1 -8976.445,E2 -8976.445} C_VEL
LIN {X 0,Y 439.44,Z 385.751,A -85,B 0,C 180,E1 -8977.531,E2 -8977.531} C_VEL
LIN {X 0,Y 439.418,Z 385.755,A -85,B 0,C 180,E1 -8980.662,E2 -8980.662} C_VEL
LIN {X 0,Y 439.439,Z 385.751,A -85,B 0,C 180,E1 -8984.224,E2 -8984.224} C_VEL
LIN {X 0,Y 439.492,Z 385.741,A -85,B 0,C 180,E1 -8988.002,E2 -8988.002} C_VEL
LIN {X 0,Y 439.525,Z 385.736,A -85,B 0,C 180,E1 -8991.726,E2 -8991.726} C_VEL
LIN {X 0,Y 439.605,Z 385.727,A -85,B 0,C 180,E1 -8994.496,E2 -8994.496} C_VEL
LIN {X 0,Y 439.614,Z 385.724,A -85,B 0,C 180,E1 -8998.168,E2 -8998.168} C_VEL
LIN {X 0,Y 439.741,Z 385.71,A -85,B 0,C 180,E1 -9000,E2 -9000} C_VEL
LIN {X 0,Y 439.642,Z 385.722,A -85,B 0,C 180,E1 -9002.749,E2 -9002.749} C_VEL
LIN {X 0,Y 439.6,Z 385.724,A -85,B 0,C 180,E1 -9006.426,E2 -9006.426} C_VEL
LIN {X 0,Y 439.48,Z 385.739,A -85,B 0,C 180,E1 -9009.202,E2 -9009.202} C_VEL
LIN {X 0,Y 439.481,Z 385.741,A -85,B 0,C 180,E1 -9012.728,E2 -9012.728} C_VEL
LIN {X 0,Y 439.438,Z 385.746,A -85,B 0,C 180,E1 -9016.356,E2 -9016.356} C_VEL
LIN {X 0,Y 439.414,Z 385.752,A -85,B 0,C 180,E1 -9019.626,E2 -9019.626} C_VEL
LIN {X 0,Y 439.359,Z 385.757,A -85,B 0,C 180,E1 -9022.576,E2 -9022.576} C_VEL
LIN {X 0,Y 439.385,Z 385.754,A -85,B 0,C 180,E1 -9025.586,E2 -9025.586} C_VEL
LIN {X 0,Y 439.405,Z 385.753,A -85,B 0,C 180,E1 -9028.675,E2 -9028.675} C_VEL
LIN {X 0,Y 439.355,Z 385.755,A -85,B 0,C 180,E1 -9031.862,E2 -9031.862} C_VEL
LIN {X 0,Y 439.383,Z 385.756,A -85,B 0,C 180,E1 -9035.158,E2 -9035.158} C_VEL
LIN {X 0,Y 439.382,Z 385.754,A -85,B 0,C 180,E1 -9038.595,E2 -9038.595} C_VEL
LIN {X 0,Y 439.389,Z 385.754,A -85,B 0,C 180,E1 -9041.262,E2 -9041.262} C_VEL
LIN {X 0,Y 439.396,Z 385.754,A -85,B 0,C 180,E1 -9044.73,E2 -9044.73} C_VEL
LIN {X 0,Y 439.399,Z 385.754,A -85,B 0,C 180,E1 -9047.8,E2 -9047.8} C_VEL
LIN {X 0,Y 439.44,Z 385.749,A -85,B 0,C 180,E1 -9050.233,E2 -9050.233} C_VEL
LIN {X 0,Y 439.393,Z 385.918,A -85,B 0,C 180,E1 -9053.718,E2 -9053.718} C_VEL
LIN {X 0,Y 440.89,Z 393.269,A -85,B 0,C 180,E1 -9056.64,E2 -9056.64} C_VEL
LIN {X 0,Y 441.996,Z 400.089,A -85,B 0,C 180,E1 -9059.164,E2 -9059.164} C_VEL
LIN {X 0,Y 441.471,Z 406.954,A -85,B 0,C 180,E1 -9061.475,E2 -9061.475} C_VEL
LIN {X 0,Y 440.635,Z 417.95,A -85,B 0,C 180,E1 -9065,E2 -9065} C_VEL
LIN {X 0,Y 439.927,Z 428.993,A -85,B 0,C 180,E1 -9068.445,E2 -9068.445} C_VEL
LIN {X 0,Y 439.375,Z 440.253,A -85,B 0,C 180,E1 -9071.828,E2 -9071.828} C_VEL
LIN {X 0,Y 439.156,Z 447.13,A -85,B 0,C 180,E1 -9073.857,E2 -9073.857} C_VEL
LIN {X 0,Y 441.06,Z 461.214,A -85,B 0,C 180,E1 -9074.3,E2 -9074.3} C_VEL
LIN {X 0,Y 441.999,Z 471.072,A -85,B 0,C 180,E1 -9074.733,E2 -9074.733} C_VEL
LIN {X 0,Y 441.468,Z 482.986,A -85,B 0,C 180,E1 -9075.364,E2 -9075.364} C_VEL
LIN {X 0,Y 440.867,Z 494.449,A -85,B 0,C 180,E1 -9076.168,E2 -9076.168} C_VEL
LIN {X 0,Y 440.304,Z 504.866,A -85,B 0,C 180,E1 -9077.09,E2 -9077.09} C_VEL
LIN {X 0,Y 439.815,Z 515.357,A -85,B 0,C 180,E1 -9078.247,E2 -9078.247} C_VEL
LIN {X 0,Y 439.189,Z 525.372,A -85,B 0,C 180,E1 -9079.631,E2 -9079.631} C_VEL
LIN {X 0,Y 438.824,Z 533.47,A -85,B 0,C 180,E1 -9081.019,E2 -9081.019} C_VEL
LIN {X 0,Y 438.606,Z 538.947,A -85,B 0,C 180,E1 -9082.174,E2 -9082.174} C_VEL
LIN {X 0,Y 438.402,Z 544.684,A -85,B 0,C 180,E1 -9083.681,E2 -9083.681} C_VEL
LIN {X 0,Y 438.399,Z 548.407,A -85,B 0,C 180,E1 -9084.944,E2 -9084.944} C_VEL
LIN {X 0,Y 438.317,Z 551.45,A -85,B 0,C 180,E1 -9086.325,E2 -9086.325} C_VEL
LIN {X 0,Y 438.373,Z 552.923,A -85,B 0,C 180,E1 -9087.245,E2 -9087.245} C_VEL
LIN {X 0,Y 438.354,Z 553.948,A -85,B 0,C 180,E1 -9088.165,E2 -9088.165} C_VEL
LIN {X 0,Y 438.308,Z 554.573,A -85,B 0,C 180,E1 -9089.083,E2 -9089.083} C_VEL
LIN {X 0,Y 438.281,Z 554.792,A -85,B 0,C 180,E1 -9090.002,E2 -9090.002} C_VEL
LIN {X 0,Y 438.309,Z 554.573,A -85,B 0,C 180,E1 -9090.921,E2 -9090.921} C_VEL
LIN {X 0,Y 438.367,Z 553.945,A -85,B 0,C 180,E1 -9091.839,E2 -9091.839} C_VEL
LIN {X 0,Y 438.374,Z 552.916,A -85,B 0,C 180,E1 -9092.759,E2 -9092.759} C_VEL
LIN {X 0,Y 438.32,Z 551.453,A -85,B 0,C 180,E1 -9093.679,E2 -9093.679} C_VEL
LIN {X 0,Y 438.401,Z 548.421,A -85,B 0,C 180,E1 -9095.06,E2 -9095.06} C_VEL
LIN {X 0,Y 438.451,Z 544.309,A -85,B 0,C 180,E1 -9096.444,E2 -9096.444} C_VEL
LIN {X 0,Y 438.669,Z 537.974,A -85,B 0,C 180,E1 -9098.06,E2 -9098.06} C_VEL
LIN {X 0,Y 438.986,Z 531.071,A -85,B 0,C 180,E1 -9099.447,E2 -9099.447} C_VEL
LIN {X 0,Y 439.365,Z 522.448,A -85,B 0,C 180,E1 -9100.835,E2 -9100.835} C_VEL
LIN {X 0,Y 439.983,Z 512.563,A -85,B 0,C 180,E1 -9102.104,E2 -9102.104} C_VEL
LIN {X 0,Y 440.419,Z 502.286,A -85,B 0,C 180,E1 -9103.173,E2 -9103.173} C_VEL
LIN {X 0,Y 441.035,Z 491.573,A -85,B 0,C 180,E1 -9104.066,E2 -9104.066} C_VEL
LIN {X 0,Y 441.713,Z 479.269,A -85,B 0,C 180,E1 -9104.868,E2 -9104.868} C_VEL
LIN {X 0,Y 441.9,Z 468.927,A -85,B 0,C 180,E1 -9105.392,E2 -9105.392} C_VEL
LIN {X 0,Y 440.458,Z 455.901,A -85,B 0,C 180,E1 -9105.931,E2 -9105.931} C_VEL
LIN {X 0,Y 439.127,Z 446.966,A -85,B 0,C 180,E1 -9106.233,E2 -9106.233} C_VEL
LIN {X 0,Y 439.577,Z 435.539,A -85,B 0,C 180,E1 -9109.62,E2 -9109.62} C_VEL
LIN {X 0,Y 440.123,Z 425.88,A -85,B 0,C 180,E1 -9112.536,E2 -9112.536} C_VEL
LIN {X 0,Y 440.745,Z 416.257,A -85,B 0,C 180,E1 -9115.503,E2 -9115.503} C_VEL
LIN {X 0,Y 441.596,Z 405.488,A -85,B 0,C 180,E1 -9118.916,E2 -9118.916} C_VEL
LIN {X 0,Y 441.872,Z 399.698,A -85,B 0,C 180,E1 -9120.809,E2 -9120.809} C_VEL
LIN {X 0,Y 440.997,Z 394.025,A -85,B 0,C 180,E1 -9122.811,E2 -9122.811} C_VEL
LIN {X 0,Y 439.66,Z 387.001,A -85,B 0,C 180,E1 -9125.389,E2 -9125.389} C_VEL
LIN {X 0,Y 439.388,Z 385.756,A -85,B 0,C 180,E1 -9125.914,E2 -9125.914} C_VEL
LIN {X 0,Y 439.368,Z 385.757,A -85,B 0,C 180,E1 -9128.598,E2 -9128.598} C_VEL
LIN {X 0,Y 439.353,Z 385.759,A -85,B 0,C 180,E1 -9132.211,E2 -9132.211} C_VEL
LIN {X 0,Y 439.38,Z 385.756,A -85,B 0,C 180,E1 -9135.268,E2 -9135.268} C_VEL
LIN {X 0,Y 439.37,Z 385.754,A -85,B 0,C 180,E1 -9138.747,E2 -9138.747} C_VEL
LIN {X 0,Y 439.372,Z 385.75,A -85,B 0,C 180,E1 -9141.61,E2 -9141.61} C_VEL
LIN {X 0,Y 439.403,Z 385.751,A -85,B 0,C 180,E1 -9144.844,E2 -9144.844} C_VEL
LIN {X 0,Y 439.375,Z 385.756,A -85,B 0,C 180,E1 -9148.139,E2 -9148.139} C_VEL
LIN {X 0,Y 439.393,Z 385.754,A -85,B 0,C 180,E1 -9151.61,E2 -9151.61} C_VEL
LIN {X 0,Y 439.358,Z 385.756,A -85,B 0,C 180,E1 -9154.412,E2 -9154.412} C_VEL
LIN {X 0,Y 439.367,Z 385.755,A -85,B 0,C 180,E1 -9157.424,E2 -9157.424} C_VEL
LIN {X 0,Y 439.448,Z 385.748,A -85,B 0,C 180,E1 -9160.663,E2 -9160.663} C_VEL
LIN {X 0,Y 439.468,Z 385.747,A -85,B 0,C 180,E1 -9164.224,E2 -9164.224} C_VEL
LIN {X 0,Y 439.487,Z 385.743,A -85,B 0,C 180,E1 -9168.001,E2 -9168.001} C_VEL
LIN {X 0,Y 439.485,Z 385.742,A -85,B 0,C 180,E1 -9171.725,E2 -9171.725} C_VEL
LIN {X 0,Y 439.601,Z 385.73,A -85,B 0,C 180,E1 -9174.495,E2 -9174.495} C_VEL
LIN {X 0,Y 439.238,Z 385.873,A -85,B 0,C 180,E1 -9176.33,E2 -9176.33} C_VEL
LIN {X 0,Y 439.547,Z 391.077,A -85,B 0,C 180,E1 -9178.625,E2 -9178.625} C_VEL
LIN {X 0,Y 439.306,Z 397.265,A -85,B 0,C 180,E1 -9181.375,E2 -9181.375} C_VEL
LIN {X 0,Y 439.179,Z 404.339,A -85,B 0,C 180,E1 -9184.589,E2 -9184.589} C_VEL
LIN {X 0,Y 439.065,Z 411.447,A -85,B 0,C 180,E1 -9187.819,E2 -9187.819} C_VEL
LIN {X 0,Y 438.894,Z 418.472,A -85,B 0,C 180,E1 -9191.078,E2 -9191.078} C_VEL
LIN {X 0,Y 438.75,Z 425.523,A -85,B 0,C 180,E1 -9194.376,E2 -9194.376} C_VEL
LIN {X 0,Y 438.736,Z 425.968,A -85,B 0,C 180,E1 -9194.583,E2 -9194.583} C_VEL
LIN {X 0,Y 441.81,Z 440.515,A -85,B 0,C 180,E1 -9195.187,E2 -9195.187} C_VEL
LIN {X 0,Y 442.786,Z 446.334,A -85,B 0,C 180,E1 -9195.477,E2 -9195.477} C_VEL
LIN {X 0,Y 442.203,Z 458.938,A -85,B 0,C 180,E1 -9196.148,E2 -9196.148} C_VEL
LIN {X 0,Y 441.61,Z 470.424,A -85,B 0,C 180,E1 -9196.95,E2 -9196.95} C_VEL
LIN {X 0,Y 441.048,Z 480.814,A -85,B 0,C 180,E1 -9197.863,E2 -9197.863} C_VEL
LIN {X 0,Y 440.406,Z 490.989,A -85,B 0,C 180,E1 -9198.974,E2 -9198.974} C_VEL
LIN {X 0,Y 439.813,Z 501.043,A -85,B 0,C 180,E1 -9200.337,E2 -9200.337} C_VEL
LIN {X 0,Y 439.342,Z 508.455,A -85,B 0,C 180,E1 -9201.587,E2 -9201.587} C_VEL
LIN {X 0,Y 438.915,Z 515.669,A -85,B 0,C 180,E1 -9203.097,E2 -9203.097} C_VEL
LIN {X 0,Y 438.625,Z 521.364,A -85,B 0,C 180,E1 -9204.619,E2 -9204.619} C_VEL
LIN {X 0,Y 438.452,Z 525.642,A -85,B 0,C 180,E1 -9206.15,E2 -9206.15} C_VEL
LIN {X 0,Y 438.279,Z 528.711,A -85,B 0,C 180,E1 -9207.712,E2 -9207.712} C_VEL
LIN {X 0,Y 438.2,Z 530.109,A -85,B 0,C 180,E1 -9208.76,E2 -9208.76} C_VEL
LIN {X 0,Y 438.151,Z 531.03,A -85,B 0,C 180,E1 -9209.982,E2 -9209.982} C_VEL
LIN {X 0,Y 438.142,Z 531.143,A -85,B 0,C 180,E1 -9211.771,E2 -9211.771} C_VEL
LIN {X 0,Y 438.198,Z 529.773,A -85,B 0,C 180,E1 -9213.487,E2 -9213.487} C_VEL
LIN {X 0,Y 438.328,Z 526.902,A -85,B 0,C 180,E1 -9215.254,E2 -9215.254} C_VEL
LIN {X 0,Y 438.523,Z 523.211,A -85,B 0,C 180,E1 -9216.742,E2 -9216.742} C_VEL
LIN {X 0,Y 438.749,Z 518.003,A -85,B 0,C 180,E1 -9218.288,E2 -9218.288} C_VEL
LIN {X 0,Y 439.046,Z 511.364,A -85,B 0,C 180,E1 -9219.814,E2 -9219.814} C_VEL
LIN {X 0,Y 439.516,Z 503.275,A -85,B 0,C 180,E1 -9221.274,E2 -9221.274} C_VEL
LIN {X 0,Y 440.081,Z 494.005,A -85,B 0,C 180,E1 -9222.612,E2 -9222.612} C_VEL
LIN {X 0,Y 440.663,Z 484.056,A -85,B 0,C 180,E1 -9223.77,E2 -9223.77} C_VEL
LIN {X 0,Y 441.268,Z 472.914,A -85,B 0,C 180,E1 -9224.81,E2 -9224.81} C_VEL
LIN {X 0,Y 441.755,Z 462.766,A -85,B 0,C 180,E1 -9225.571,E2 -9225.571} C_VEL
LIN {X 0,Y 442.362,Z 450.904,A -85,B 0,C 180,E1 -9226.268,E2 -9226.268} C_VEL
LIN {X 0,Y 442.45,Z 445.116,A -85,B 0,C 180,E1 -9226.546,E2 -9226.546} C_VEL
LIN {X 0,Y 439.988,Z 431.855,A -85,B 0,C 180,E1 -9227.126,E2 -9227.126} C_VEL
LIN {X 0,Y 438.708,Z 425.435,A -85,B 0,C 180,E1 -9227.373,E2 -9227.373} C_VEL
LIN {X 0,Y 438.812,Z 418.245,A -85,B 0,C 180,E1 -9230.799,E2 -9230.799} C_VEL
LIN {X 0,Y 438.951,Z 411.036,A -85,B 0,C 180,E1 -9234.239,E2 -9234.239} C_VEL
LIN {X 0,Y 439.115,Z 404.052,A -85,B 0,C 180,E1 -9237.566,E2 -9237.566} C_VEL
LIN {X 0,Y 439.242,Z 397.29,A -85,B 0,C 180,E1 -9240.789,E2 -9240.789} C_VEL
LIN {X 0,Y 439.364,Z 389.685,A -85,B 0,C 180,E1 -9244.411,E2 -9244.411} C_VEL
LIN {X 0,Y 439.512,Z 385.74,A -85,B 0,C 180,E1 -9246.33,E2 -9246.33} C_VEL
LIN {X 0,Y 439.39,Z 385.753,A -85,B 0,C 180,E1 -9249.396,E2 -9249.396} C_VEL
LIN {X 0,Y 439.426,Z 385.749,A -85,B 0,C 180,E1 -9252.308,E2 -9252.308} C_VEL
LIN {X 0,Y 439.449,Z 385.749,A -85,B 0,C 180,E1 -9255.172,E2 -9255.172} C_VEL
LIN {X 0,Y 439.451,Z 385.744,A -85,B 0,C 180,E1 -9258.36,E2 -9258.36} C_VEL
LIN {X 0,Y 438.774,Z 385.83,A -85,B 0,C 180,E1 -9259.125,E2 -9259.125} C_VEL
LIN {X 0,Y 435.986,Z 386.177,A -85,B 0,C 180,E1 -9260.369,E2 -9260.369} C_VEL
LIN {X 0,Y 433.631,Z 386.473,A -85,B 0,C 180,E1 -9261.372,E2 -9261.372} C_VEL
LIN {X 0,Y 432.605,Z 386.598,A -85,B 0,C 180,E1 -9262.147,E2 -9262.147} C_VEL
LIN {X 0,Y 432.512,Z 386.61,A -85,B 0,C 180,E1 -9262.409,E2 -9262.409} C_VEL
LIN {X 0,Y 432.584,Z 386.605,A -85,B 0,C 180,E1 -9264.404,E2 -9264.404} C_VEL
LIN {X 0,Y 432.596,Z 386.601,A -85,B 0,C 180,E1 -9268.136,E2 -9268.136} C_VEL
LIN {X 0,Y 432.677,Z 386.647,A -85,B 0,C 180,E1 -9269.3,E2 -9269.3} C_VEL
LIN {X 0,Y 432.738,Z 389.36,A -85,B 0,C 180,E1 -9270.928,E2 -9270.928} C_VEL
LIN {X 0,Y 432.338,Z 395.739,A -85,B 0,C 180,E1 -9274.66,E2 -9274.66} C_VEL
LIN {X 0,Y 432.239,Z 400.606,A -85,B 0,C 180,E1 -9277.472,E2 -9277.472} C_VEL
LIN {X 0,Y 431.977,Z 407.309,A -85,B 0,C 180,E1 -9281.256,E2 -9281.256} C_VEL
LIN {X 0,Y 431.739,Z 412.463,A -85,B 0,C 180,E1 -9284.131,E2 -9284.131} C_VEL
LIN {X 0,Y 431.591,Z 417.738,A -85,B 0,C 180,E1 -9287.042,E2 -9287.042} C_VEL
LIN {X 0,Y 431.528,Z 422.502,A -85,B 0,C 180,E1 -9289.635,E2 -9289.635} C_VEL
LIN {X 0,Y 433.68,Z 434.144,A -85,B 0,C 180,E1 -9290.14,E2 -9290.14} C_VEL
LIN {X 0,Y 434.561,Z 440.118,A -85,B 0,C 180,E1 -9290.468,E2 -9290.468} C_VEL
LIN {X 0,Y 434.113,Z 450.493,A -85,B 0,C 180,E1 -9291.111,E2 -9291.111} C_VEL
LIN {X 0,Y 433.557,Z 460.096,A -85,B 0,C 180,E1 -9291.888,E2 -9291.888} C_VEL
LIN {X 0,Y 433.164,Z 468.755,A -85,B 0,C 180,E1 -9292.77,E2 -9292.77} C_VEL
LIN {X 0,Y 432.695,Z 477.921,A -85,B 0,C 180,E1 -9293.955,E2 -9293.955} C_VEL
LIN {X 0,Y 432.311,Z 484.425,A -85,B 0,C 180,E1 -9295.001,E2 -9295.001} C_VEL
LIN {X 0,Y 432.057,Z 489.738,A -85,B 0,C 180,E1 -9296.049,E2 -9296.049} C_VEL
LIN {X 0,Y 431.744,Z 494.14,A -85,B 0,C 180,E1 -9297.113,E2 -9297.113} C_VEL
LIN {X 0,Y 431.57,Z 498.382,A -85,B 0,C 180,E1 -9298.433,E2 -9298.433} C_VEL
LIN {X 0,Y 431.506,Z 500.41,A -85,B 0,C 180,E1 -9299.246,E2 -9299.246} C_VEL
LIN {X 0,Y 431.339,Z 502.483,A -85,B 0,C 180,E1 -9300.335,E2 -9300.335} C_VEL
LIN {X 0,Y 431.171,Z 504.347,A -85,B 0,C 180,E1 -9302.05,E2 -9302.05} C_VEL
LIN {X 0,Y 431.197,Z 504.548,A -85,B 0,C 180,E1 -9303.774,E2 -9303.774} C_VEL
LIN {X 0,Y 431.324,Z 503.146,A -85,B 0,C 180,E1 -9305.443,E2 -9305.443} C_VEL
LIN {X 0,Y 431.506,Z 500.234,A -85,B 0,C 180,E1 -9307.054,E2 -9307.054} C_VEL
LIN {X 0,Y 431.799,Z 495.822,A -85,B 0,C 180,E1 -9308.625,E2 -9308.625} C_VEL
LIN {X 0,Y 432.043,Z 491.501,A -85,B 0,C 180,E1 -9309.768,E2 -9309.768} C_VEL
LIN {X 0,Y 432.402,Z 484.748,A -85,B 0,C 180,E1 -9311.163,E2 -9311.163} C_VEL
LIN {X 0,Y 432.874,Z 476.233,A -85,B 0,C 180,E1 -9312.513,E2 -9312.513} C_VEL
LIN {X 0,Y 433.432,Z 467.481,A -85,B 0,C 180,E1 -9313.59,E2 -9313.59} C_VEL
LIN {X 0,Y 434.022,Z 457.443,A -85,B 0,C 180,E1 -9314.563,E2 -9314.563} C_VEL
LIN {X 0,Y 434.532,Z 446.699,A -85,B 0,C 180,E1 -9315.364,E2 -9315.364} C_VEL
LIN {X 0,Y 434.638,Z 438.883,A -85,B 0,C 180,E1 -9315.821,E2 -9315.821} C_VEL
LIN {X 0,Y 432.529,Z 427.276,A -85,B 0,C 180,E1 -9316.406,E2 -9316.406} C_VEL
LIN {X 0,Y 431.585,Z 422.911,A -85,B 0,C 180,E1 -9316.608,E2 -9316.608} C_VEL
LIN {X 0,Y 431.689,Z 416.968,A -85,B 0,C 180,E1 -9319.917,E2 -9319.917} C_VEL
LIN {X 0,Y 431.86,Z 411.527,A -85,B 0,C 180,E1 -9322.978,E2 -9322.978} C_VEL
LIN {X 0,Y 432.034,Z 406.119,A -85,B 0,C 180,E1 -9326.055,E2 -9326.055} C_VEL
LIN {X 0,Y 432.273,Z 400.198,A -85,B 0,C 180,E1 -9329.5,E2 -9329.5} C_VEL
LIN {X 0,Y 432.55,Z 394.33,A -85,B 0,C 180,E1 -9332.939,E2 -9332.939} C_VEL
LIN {X 0,Y 432.661,Z 389.173,A -85,B 0,C 180,E1 -9336.041,E2 -9336.041} C_VEL
LIN {X 0,Y 432.377,Z 386.631,A -85,B 0,C 180,E1 -9337.758,E2 -9337.758} C_VEL
LIN {X 0,Y 432.363,Z 386.634,A -85,B 0,C 180,E1 -9341.029,E2 -9341.029} C_VEL
LIN {X 0,Y 432.406,Z 386.627,A -85,B 0,C 180,E1 -9343.961,E2 -9343.961} C_VEL
LIN {X 0,Y 432.463,Z 386.617,A -85,B 0,C 180,E1 -9347.804,E2 -9347.804} C_VEL
LIN {X 0,Y 432.469,Z 386.616,A -85,B 0,C 180,E1 -9351.59,E2 -9351.59} C_VEL
LIN {X 0,Y 432.581,Z 386.603,A -85,B 0,C 180,E1 -9354.406,E2 -9354.406} C_VEL
LIN {X 0,Y 432.584,Z 386.6,A -85,B 0,C 180,E1 -9358.138,E2 -9358.138} C_VEL
LIN {X 0,Y 432.711,Z 386.585,A -85,B 0,C 180,E1 -9360,E2 -9360} C_VEL
LIN {X 0,Y 432.591,Z 386.6,A -85,B 0,C 180,E1 -9362.794,E2 -9362.794} C_VEL
LIN {X 0,Y 432.553,Z 386.601,A -85,B 0,C 180,E1 -9366.531,E2 -9366.531} C_VEL
LIN {X 0,Y 432.424,Z 386.618,A -85,B 0,C 180,E1 -9369.354,E2 -9369.354} C_VEL
LIN {X 0,Y 432.422,Z 386.62,A -85,B 0,C 180,E1 -9372.813,E2 -9372.813} C_VEL
LIN {X 0,Y 432.401,Z 386.623,A -85,B 0,C 180,E1 -9376.485,E2 -9376.485} C_VEL
LIN {X 0,Y 432.361,Z 386.629,A -85,B 0,C 180,E1 -9379.96,E2 -9379.96} C_VEL
LIN {X 0,Y 432.309,Z 386.636,A -85,B 0,C 180,E1 -9382.965,E2 -9382.965} C_VEL
LIN {X 0,Y 432.344,Z 386.632,A -85,B 0,C 180,E1 -9386.034,E2 -9386.034} C_VEL
LIN {X 0,Y 432.333,Z 386.63,A -85,B 0,C 180,E1 -9389.189,E2 -9389.189} C_VEL
LIN {X 0,Y 432.307,Z 386.633,A -85,B 0,C 180,E1 -9392.295,E2 -9392.295} C_VEL
LIN {X 0,Y 432.323,Z 386.633,A -85,B 0,C 180,E1 -9394.679,E2 -9394.679} C_VEL
LIN {X 0,Y 432.336,Z 386.635,A -85,B 0,C 180,E1 -9398.15,E2 -9398.15} C_VEL
